DATA_BLOCK "DB22_DisplayData"   // DB22
{ S7_Optimized_Access := 'FALSE' }
AUTHOR : Robopac
VERSION : 0.0
// stored: AutoNumber false, IsOnlyStoredInLoadMemory false, IsWriteProtectedInAS false
   VAR RETAIN
      dbx0_0 : Bool := FALSE;   // Technoplat manual(Display): Table rotation forward
      dbx0_1 : Bool := FALSE;   // Technoplat manual(Display): Spool carriage upward
      dbx0_2 : Bool := FALSE;   // Technoplat manual(Display): Spool carriage downward
      dbx0_3 : Bool := FALSE;   // Technoplat manual(Display): Pressure plate upward/downward
      dbx0_4 : Bool := FALSE;   // Technoplat manual(Display): Pallet lifter upward/downward
      dbx0_5 : Bool := FALSE;   // Technoplat manual(Display): Rope unit open/close
      dbx0_6 : Bool := FALSE;   // Technoplat manual(Display): Prestretch
      dbx0_7 : Bool := FALSE;   // Technoplat manual(Display): Spool carriage to film broken position
      dbx1_0 : Bool := FALSE;   // Clamp manual(Display): Clamp upward/downward
      dbx1_1 : Bool := FALSE;   // Clamp manual(Display): Welder unit upward/downward
      dbx1_2 : Bool := FALSE;   // Clamp manual(Display): Welder contrast upward/downward
      dbx1_3 : Bool := FALSE;   // Clamp manual(Display): Clamp carriage forward/backward
      dbx1_4 : Bool := FALSE;   // Clamp manual(Display): Clamp open/close
      dbx1_5 : Bool := FALSE;   // Clamp manual(Display): Cut and welder arm forward/backward
      dbx1_6 : Bool := FALSE;   // Clamp manual(Display): Welder unit forward/backward
      dbx1_7 : Bool := FALSE;   // Clamp manual(Display):
      dbx2_0 : Bool := FALSE;   // Top manual(Display): Top carriage upward
      dbx2_1 : Bool := FALSE;   // Top manual(Display): Top carriage downward
      dbx2_2 : Bool := FALSE;   // Top manual(Display): Top carriage forward
      dbx2_3 : Bool := FALSE;   // Top manual(Display): Top carriage backward
      dbx2_4 : Bool := FALSE;   // Top manual(Display): Opening/closing clamp to pull top film
      dbx2_5 : Bool := FALSE;   // Top manual(Display): Opening/closing clamp to block top film
      dbx2_6 : Bool := FALSE;   // Top manual(Display): Top film cutter forward/backward
      dbx2_7 : Bool := FALSE;   // Top manual(Display): Arm rotation to phase 2 sensor for top
      dbx3_0 : Bool := FALSE;   // Technoplat manual (Display): Rotation to unload
      dbx3_1 : Bool := FALSE;   // Technoplat manual (Display): Rotation to 0
      dbx3_2 : Bool := FALSE;   // Technoplat manual (Display): Rotation to load
      dbx3_3 : Bool := FALSE;
      dbx3_4 : Bool := FALSE;   // Technoplat manual(Display): Rope unit lower open/close
      dbx3_5 : Bool := FALSE;
      dbx3_6 : Bool := FALSE;
      dbx3_7 : Bool := FALSE;
      dbx4_0 : Bool := FALSE;   // Conveyor manual(Display): CMD PRESSED
      dbx4_1 : Bool := FALSE;   // Conveyor manual(Display): Load CM [p18]
      dbx4_2 : Bool := FALSE;   // Conveyor manual(Display): Unload CM [p18]
      dbx4_3 : Bool := FALSE;   // Conveyor manual(Display): RESET ENCODER
      dbx4_4 : Bool := FALSE;   // Conveyor manual(Display): Load CM [Sysdata]
      dbx4_5 : Bool := FALSE;   // Conveyor manual(Display): [not used]
      dbx4_6 : Bool := FALSE;   // Conveyor manual(Display): CM backward slow
      dbx4_7 : Bool := FALSE;   // Conveyor manual(Display): CM forward slow
      dbb5 : Byte := 16#09;   // Conveyor manual operation
      dbx6_0 : Bool := FALSE;   // Manual Signal(Display): Pallet ready in infeed (Input)
      dbx6_1 : Bool := FALSE;   // Manual Signal(Display): Ready to receive pallet infeed (Output)
      dbx6_2 : Bool := FALSE;   // Manual Signal(Display): End of transfer pallet infeed (Output)
      dbx6_3 : Bool := FALSE;   // Manual Signal(Display): Pallet ready in outfeed (Output)
      dbx6_4 : Bool := FALSE;   // Manual Signal(Display): Ready to receive pallet outfeed (Input)
      dbx6_5 : Bool := FALSE;   // Manual Signal(Display): End of transfer pallet outfeed (Input)
      dbx6_6 : Bool := FALSE;   // Manual Signal(Display): Start wrapping signal (Input)
      dbx6_7 : Bool := FALSE;   // Manual Signal(Display): Customer conveyor stopped signal (Input)
      dbx7_0 : Bool := FALSE;   // Manual Signal(Display): Machine in position signal (Output)
      dbx7_1 : Bool := FALSE;   // Manual Signal(Display): Wrapp ended signal (Output)
      dbx7_2 : Bool := FALSE;   // Manual Signal(Display): Pallet in position for label
      dbx7_3 : Bool := TRUE;   // Manual Signal(Display): Label arm in position for pallet transfer
      dbx7_4 : Bool := FALSE;   // Manual Signal(Display): Label cycle ended
      dbx7_5 : Bool := FALSE;   // Manual Signal(Display): Label fault
      dbx7_6 : Bool := FALSE;
      dbx7_7 : Bool := FALSE;
      dbw8 : Int := 0;
      dbw10 : Int := 0;
      dbw12 : Int := 0;
      dbx14_0 : Bool := FALSE;   // Technoplat manual(Program): Table rotation forward
      dbx14_1 : Bool := FALSE;   // Technoplat manual(Program): Spool carriage upward
      dbx14_2 : Bool := FALSE;   // Technoplat manual(Program): Spool carriage downward
      dbx14_3 : Bool := FALSE;   // Technoplat manual(Program): Pressure plate downward
      dbx14_4 : Bool := FALSE;   // Technoplat manual(Program): Pressure plate upward
      dbx14_5 : Bool := FALSE;   // Technoplat manual(Program): Pallet lifter upward
      dbx14_6 : Bool := FALSE;   // Technoplat manual(Program): Pallet lifter downward
      dbx14_7 : Bool := FALSE;   // Technoplat manual(Program): Rope unit closing
      dbx15_0 : Bool := FALSE;   // Technoplat manual(Program): Rope unit opening
      dbx15_1 : Bool := FALSE;   // Technoplat manual(Program): Prestretch
      dbx15_2 : Bool := FALSE;   // Technoplat manual(Program): Spool carriage to film broken position
      dbx15_3 : Bool := FALSE;   // Technoplat manual(Program): Rope unit Lower closing
      dbx15_4 : Bool := FALSE;   // Technoplat manual(Program): Rope unit Lower opening
      dbx15_5 : Bool := FALSE;   // Technoplat manual(Program): CM Backward slow
      dbx15_6 : Bool := FALSE;   // Technoplat manual(Program): CM Forward slow
      dbx15_7 : Bool := FALSE;   // Technoplat manual(Program):
      dbx16_0 : Bool := FALSE;   // Clamp manual(Program): Clamp upward
      dbx16_1 : Bool := FALSE;   // Clamp manual(Program): Clamp downward
      dbx16_2 : Bool := FALSE;   // Clamp manual(Program): Welder unit upward
      dbx16_3 : Bool := FALSE;   // Clamp manual(Program): Welder unit downward
      dbx16_4 : Bool := FALSE;   // Clamp manual(Program): Welder contrast upward
      dbx16_5 : Bool := FALSE;   // Clamp manual(Program): Welder contrast downward
      dbx16_6 : Bool := FALSE;   // Clamp manual(Program): Clamp carriage forward
      dbx16_7 : Bool := FALSE;   // Clamp manual(Program): Clamp carriage backward
      dbx17_0 : Bool := FALSE;   // Clamp manual(Program): Clamp open
      dbx17_1 : Bool := FALSE;   // Clamp manual(Program): Clamp close
      dbx17_2 : Bool := FALSE;   // Clamp manual(Program): Cut and welder arm forward
      dbx17_3 : Bool := FALSE;   // Clamp manual(Program): Cut and welder arm backward
      dbx17_4 : Bool := FALSE;   // Clamp manual(Program): Welder unit forward
      dbx17_5 : Bool := FALSE;   // Clamp manual(Program): Welder unit backward
      dbx17_6 : Bool := FALSE;   // Clamp manual(Program):
      dbx17_7 : Bool := FALSE;   // Clamp manual(Program):
      dbx18_0 : Bool := FALSE;   // Top manual(Program): Top carriage upward
      dbx18_1 : Bool := FALSE;   // Top manual(Program): Top carriage downward
      dbx18_2 : Bool := FALSE;   // Top manual(Program): Top carriage forward
      dbx18_3 : Bool := FALSE;   // Top manual(Program): Top carriage backward
      dbx18_4 : Bool := FALSE;   // Top manual(Program): Opening clamp to pull top film
      dbx18_5 : Bool := FALSE;   // Top manual(Program): Closing clamp to pull top film
      dbx18_6 : Bool := FALSE;   // Top manual(Program): Opening clamp to block top film
      dbx18_7 : Bool := FALSE;   // Top manual(Program): Closing clamp to block top film
      dbx19_0 : Bool := FALSE;   // Top manual(Program): Top film cutter forward/backward
      dbx19_1 : Bool := FALSE;   // Top manual(Program): Arm rotation to phase 2 sensor for top
      dbx19_2 : Bool := FALSE;   // Technoplat manual(Program): Rotation to unload
      dbx19_3 : Bool := FALSE;   // Technoplat manual(Program): Rotation to 0
      dbx19_4 : Bool := FALSE;   // Technoplat manual(Program): Rotation to load
      dbx19_5 : Bool := FALSE;   // Top manual(Program):
      dbx19_6 : Bool := FALSE;   // Top manual(Program):
      dbx19_7 : Bool := FALSE;   // Top manual(Program):
      dbx20_0 : Bool := FALSE;   // Conveyor manual(Program): Load CM
      dbx20_1 : Bool := FALSE;   // Conveyor manual(Program): Unload CM
      dbx20_2 : Bool := FALSE;   // Conveyor manual(Program): CM backward
      dbx20_3 : Bool := FALSE;   // Conveyor manual(Program): Pos.1
      dbx20_4 : Bool := FALSE;   // Conveyor manual(Program): Pos.2
      dbx20_5 : Bool := FALSE;   // Conveyor manual(Program): Pos.3
      dbx20_6 : Bool := FALSE;   // Conveyor manual(Program): Pos.4
      dbx20_7 : Bool := FALSE;   // Conveyor manual(Program): Pos.5
      dbx21_0 : Bool := FALSE;   // Conveyor manual(Program): Pos.6
      dbx21_1 : Bool := FALSE;   // Conveyor manual(Program): Pos.7
      dbx21_2 : Bool := FALSE;   // Conveyor manual(Program): Pos.8
      dbx21_3 : Bool := FALSE;   // Conveyor manual(Program):
      dbx21_4 : Bool := FALSE;   // Conveyor manual(Program):
      dbx21_5 : Bool := FALSE;   // Conveyor manual(Program):
      dbx21_6 : Bool := FALSE;   // Conveyor manual(Program):
      dbx21_7 : Bool := FALSE;   // Conveyor manual(Program):
      dbx22_0 : Bool := FALSE;   // Manual Signal(Program): Pallet ready in infeed (Input)
      dbx22_1 : Bool := FALSE;   // Manual Signal(Program): Ready to receive pallet infeed (Output)
      dbx22_2 : Bool := FALSE;   // Manual Signal(Program): End of transfer pallet infeed (Output)
      dbx22_3 : Bool := FALSE;   // Manual Signal(Program): Pallet ready in outfeed (Output)
      dbx22_4 : Bool := FALSE;   // Manual Signal(Program): Ready to receive pallet outfeed (Input)
      dbx22_5 : Bool := FALSE;   // Manual Signal(Program): End of transfer pallet outfeed (Input)
      dbx22_6 : Bool := FALSE;   // Manual Signal(Program): Start wrapping (Input)
      dbx22_7 : Bool := FALSE;   // Manual Signal(Program): Customer conveyor stopped (Input)
      dbx23_0 : Bool := FALSE;   // Manual Signal(Program): Machine in position (Output)
      dbx23_1 : Bool := FALSE;   // Manual Signal(Program): Wrapp ended (Output)
      dbx23_2 : Bool := FALSE;   // Manual Signal(Program): Pallet ready for label
      dbx23_3 : Bool := TRUE;   // Manual Signal(Program): Label arm in position for pallet transfer
      dbx23_4 : Bool := FALSE;   // Manual Signal(Program): Label cycle ended
      dbx23_5 : Bool := FALSE;   // Manual Signal(Program): Label fault
      dbx23_6 : Bool := FALSE;
      dbx23_7 : Bool := FALSE;
      dbw24 : Int := 0;
      dbw26 : Int := 0;
      dbw28 : Int := 0;
      dbw30 : Int := 0;
      dbx32_0 : Bool := TRUE;   // Manual(Toggle bit): Pressure plate upward/downward (Technplat)
      dbx32_1 : Bool := TRUE;   // Manual(Toggle bit): Pallet lifter upward/downward (Technplat)
      dbx32_2 : Bool := FALSE;   // Manual(Toggle bit): Clamp upward/downward (Clamp)
      dbx32_3 : Bool := FALSE;   // Manual(Toggle bit): Welder unit upward/downward (Clamp)
      dbx32_4 : Bool := TRUE;   // Manual(Toggle bit): Welder contrast upward/downward (Clamp)
      dbx32_5 : Bool := FALSE;   // Manual(Toggle bit): Rope unit open/close (Technplat)
      dbx32_6 : Bool := FALSE;   // Manual(Toggle bit): Clamp open/close (Clamp)
      dbx32_7 : Bool := FALSE;   // Manual(Toggle bit): Cut and welder arm forward/backward (Clamp)
      dbx33_0 : Bool := TRUE;   // Manual(Toggle bit): Opening/closing clamp to pull top film (Top)
      dbx33_1 : Bool := TRUE;   // Manual(Toggle bit): Opening/closing clamp to block top film (Top)
      dbx33_2 : Bool := TRUE;   // Manual(Toggle bit): Welder unit forward/backward (Clamp)
      dbx33_3 : Bool := FALSE;   // Manual(Toggle bit): Clamp carriage forward/backward (Clamp)
      dbx33_4 : Bool := FALSE;   // Manual(Toggle bit): Rope unit lower open/close (Technplat)
      dbx33_5 : Bool := FALSE;   // Manual(Toggle bit):
      dbx33_6 : Bool := FALSE;   // Manual(Toggle bit):
      dbx33_7 : Bool := FALSE;   // Manual(Toggle bit):
      dbw34 : Int := 0;
      dbw36 : Int := 0;
      dbx38_0 : Bool := FALSE;   // Diagnostic signal conveyor: Pallet ready in infeed (input)
      dbx38_1 : Bool := TRUE;   // Diagnostic signal conveyor: Ready to receive pallet infeed (Output)
      dbx38_2 : Bool := FALSE;   // Diagnostic signal conveyor: End of transfer pallet infeed (Output)
      dbx38_3 : Bool := FALSE;   // Diagnostic signal conveyor: Ready to receive pallet in outfeed (Input)
      dbx38_4 : Bool := FALSE;   // Diagnostic signal conveyor: End of transfer pallet outfeed (Input)
      dbx38_5 : Bool := FALSE;   // Diagnostic signal conveyor: Pallet ready in outfeed (Output)
      dbx38_6 : Bool := FALSE;   // Diagnostic signal conveyor: Start wrapping (Input)
      dbx38_7 : Bool := FALSE;   // Diagnostic signal conveyor: Customer conveyor stopped (Input)
      dbx39_0 : Bool := FALSE;   // Diagnostic signal conveyor: Machine in position (Output)
      dbx39_1 : Bool := FALSE;   // Diagnostic signal conveyor: Wrapp ended (Output)
      dbx39_2 : Bool := FALSE;   // Diagnostic signal conveyor: Pallet ready for label
      dbx39_3 : Bool := TRUE;   // Diagnostic signal conveyor: Label arm in position for pallet transit
      dbx39_4 : Bool := FALSE;   // Diagnostic signal conveyor: Label cycle ended
      dbx39_5 : Bool := FALSE;   // Diagnostic signal conveyor: Label fault
      dbw40 : Int := 1;   // Machine status
      dbd42 : DInt := 4;   // Worked hours
      dbd46 : DInt := 95;   // Partial counter for wrapped pallet
      dbd50 : DInt := 163;   // Counter for wrapped pallet
      dbd54 : DInt := 0;
      dbw58 : Int := 21;   // Seconds for worked hours counter
      dbw60 : Int := 36;   // Minutes for worked hours counter
      dbw62 : Int := 0;   // Arm rotation speed (rpm)
      dbw64 : Int := 0;   // Arm rotation speed (rpm)
      dbw66 : Int := 15;   // Number of revolution done on last pallet
      dbw68 : Int := 777;   // Wrapping cycle time
      dbw70 : Int := 22482;   // Wrapping cycle + pallet transfer time
      dbw72 : Int := 10;   // Pallet per hour (Productivity)
      dbw74 : Int := 0;   // Film weight every wrapping cycle (g*10)
      dbw76 : Int := 0;   // Film force for film weight value
      dbw78 : Int := 0;   // Film prestretch for film weight value
      dbw80 : Int := 0;
      dbw82 : Int := 0;
      dbw84 : Int := 0;
      dbw86 : Int := 0;
      dbw88 : Int := 0;
      dbw90 : Int := 0;
      dbw92 : Int := 0;
      dbw94 : Int := 0;
      dbw96 : Int := 0;
      dbw98 : Int := 0;
   END_VAR
BEGIN
END_DATA_BLOCK

DATA_BLOCK "DB235_Program15"   // DB235
{ S7_Optimized_Access := 'FALSE' }
AUTHOR : Robopac
VERSION : 0.0
// stored: AutoNumber false, IsOnlyStoredInLoadMemory false, IsWriteProtectedInAS false
   VAR RETAIN
      Program15 { S7_SetPoint := 'True'} : "DatiProgramma";
   END_VAR
BEGIN
   Program15.Wrapping := TRUE;
   Program15.TopLenght := 500;
   Program15.TopRelease := 0;
   Program15.TopDown := 0;
   Program15.Top := 4;
   Program15.PressurePTime := 0;
   Program15.LifterTime := 0;
   Program15.RevOverContrast := 1;
   Program15.RopeEndCycle := 16#02;
   Program15.Spare4 := 16#01;
   Program15.RopeTime := 1500;
   Program15.RevOverClamp := 1;
   Program15.FilmForceFinalRev := 10;
   Program15.FilmPrestretchFinalRev := 100;
   Program15.ArmSpeed := 100;
   Program15.CarriageDown4Top := 500;
   Program15.TopDownTime := 1500;
   Program15.LapsUnderTop := 0;
   Program15.Spare6 := 0;
   Program15.Spare7 := 0;
   Program15.Spare8 := 0;
   Program15.Spare9 := 0;
   Program15.Spare10 := 0;
   Program15.Spare11 := 0;
   Program15.Spare12 := 0;
   Program15.Overlap0_1 := 0;
   Program15.Height1 := 130;
   Program15.Landmark1 := FALSE;
   Program15.Lifter1 := FALSE;
   Program15.SpareBit1H1 := FALSE;
   Program15.Airblower1 := TRUE;
   Program15.NextStep1 := TRUE;
   Program15.PressureP1 := TRUE;
   Program15.SpareByte2H1 := 16#00;
   Program15.Revolution1 := 1;
   Program15.RopeUnit1_1 := 16#01;
   Program15.RopeUnit1_2 := 16#01;
   Program15.FilmForce1 := 5;
   Program15.FilmPrestretch1 := 200;
   Program15.Spare3H1 := 0;
   Program15.Spare49 := 0;
   Program15.Spare50 := 0;
   Program15.Spare51 := 0;
   Program15.Spare52 := 0;
   Program15.Spare53 := 0;
   Program15.Overlap1_2 := 0;
   Program15.Height2 := 50;
   Program15.Landmark2 := FALSE;
   Program15.Lifter2 := FALSE;
   Program15.SpareBit1H2 := FALSE;
   Program15.Airblower2 := TRUE;
   Program15.NextStep2 := TRUE;
   Program15.PressureP2 := TRUE;
   Program15.SpareByte2H2 := 16#00;
   Program15.Revolution2 := 1;
   Program15.RopeUnit2_1 := 16#01;
   Program15.RopeUnit2_2 := 16#01;
   Program15.FilmForce2 := 20;
   Program15.FilmPrestretch2 := 200;
   Program15.Spare3H2 := 0;
   Program15.Spare54 := 0;
   Program15.Spare55 := 0;
   Program15.Spare56 := 0;
   Program15.Spare57 := 0;
   Program15.Spare58 := 0;
   Program15.Overlap2_3 := 100;
   Program15.Height3 := -50;
   Program15.Landmark3 := TRUE;
   Program15.Lifter3 := FALSE;
   Program15.SpareBit1H3 := FALSE;
   Program15.Airblower3 := TRUE;
   Program15.NextStep3 := TRUE;
   Program15.PressureP3 := TRUE;
   Program15.SpareByte2H3 := 16#00;
   Program15.Revolution3 := 2;
   Program15.RopeUnit3_1 := 16#01;
   Program15.RopeUnit3_2 := 16#01;
   Program15.FilmForce3 := 30;
   Program15.FilmPrestretch3 := 200;
   Program15.Spare3H3 := 0;
   Program15.Spare59 := 0;
   Program15.Spare60 := 0;
   Program15.Spare61 := 380;
   Program15.Spare62 := 2800;
   Program15.Spare63 := 0;
   Program15.Overlap3_4 := 100;
   Program15.Height4 := 100;
   Program15.Landmark4 := FALSE;
   Program15.Lifter4 := FALSE;
   Program15.SpareBit1H4 := FALSE;
   Program15.Airblower4 := TRUE;
   Program15.NextStep4 := TRUE;
   Program15.PressureP4 := TRUE;
   Program15.SpareByte2H4 := 16#00;
   Program15.Revolution4 := 3;
   Program15.RopeUnit4_1 := 16#02;
   Program15.RopeUnit4_2 := 16#02;
   Program15.FilmForce4 := 30;
   Program15.FilmPrestretch4 := 200;
   Program15.Spare3H4 := 0;
   Program15.Spare64 := 0;
   Program15.Spare65 := 0;
   Program15.Spare66 := 0;
   Program15.Spare67 := 0;
   Program15.Spare68 := 0;
   Program15.Overlap4_5 := 0;
   Program15.Height5 := 50;
   Program15.Landmark5 := FALSE;
   Program15.Lifter5 := FALSE;
   Program15.SpareBit1H5 := FALSE;
   Program15.Airblower5 := TRUE;
   Program15.NextStep5 := FALSE;
   Program15.PressureP5 := FALSE;
   Program15.SpareByte2H5 := 16#00;
   Program15.Revolution5 := 1;
   Program15.RopeUnit5_1 := 16#01;
   Program15.RopeUnit5_2 := 16#01;
   Program15.FilmForce5 := 30;
   Program15.FilmPrestretch5 := 200;
   Program15.Spare3H5 := 0;
   Program15.Spare69 := 0;
   Program15.Spare70 := 0;
   Program15.Spare71 := 0;
   Program15.Spare72 := 0;
   Program15.Spare73 := 0;
   Program15.Overlap5_6 := 100;
   Program15.Height6 := 50;
   Program15.Landmark6 := FALSE;
   Program15.Lifter6 := FALSE;
   Program15.SpareBit1H6 := FALSE;
   Program15.Airblower6 := TRUE;
   Program15.NextStep6 := FALSE;
   Program15.PressureP6 := FALSE;
   Program15.SpareByte2H6 := 16#00;
   Program15.Revolution6 := 2;
   Program15.RopeUnit6_1 := 16#02;
   Program15.RopeUnit6_2 := 16#01;
   Program15.FilmForce6 := 20;
   Program15.FilmPrestretch6 := 200;
   Program15.Spare3H6 := 0;
   Program15.Spare74 := 0;
   Program15.Spare75 := 0;
   Program15.Spare76 := 0;
   Program15.Spare77 := 0;
   Program15.Spare78 := 0;
   Program15.Overlap6_7 := 0;
   Program15.Height7 := 0;
   Program15.Landmark7 := FALSE;
   Program15.Lifter7 := FALSE;
   Program15.SpareBit1H7 := FALSE;
   Program15.Airblower7 := FALSE;
   Program15.NextStep7 := TRUE;
   Program15.PressureP7 := FALSE;
   Program15.SpareByte2H7 := 16#00;
   Program15.Revolution7 := 1;
   Program15.RopeUnit7_1 := 16#01;
   Program15.RopeUnit7_2 := 16#01;
   Program15.FilmForce7 := 0;
   Program15.FilmPrestretch7 := 100;
   Program15.Spare3H7 := 0;
   Program15.Spare79 := 0;
   Program15.Spare80 := 0;
   Program15.Spare81 := 0;
   Program15.Spare82 := 0;
   Program15.Spare83 := 0;
   Program15.Overlap7_8 := 0;
   Program15.Height8 := 0;
   Program15.Landmark8 := FALSE;
   Program15.Lifter8 := FALSE;
   Program15.SpareBit1H8 := FALSE;
   Program15.Airblower8 := FALSE;
   Program15.NextStep8 := TRUE;
   Program15.PressureP8 := FALSE;
   Program15.SpareByte2H8 := 16#00;
   Program15.Revolution8 := 1;
   Program15.RopeUnit8_1 := 16#01;
   Program15.RopeUnit8_2 := 16#01;
   Program15.FilmForce8 := 0;
   Program15.FilmPrestretch8 := 100;
   Program15.Spare3H8 := 0;
   Program15.Spare84 := 0;
   Program15.Spare85 := 0;
   Program15.Spare86 := 0;
   Program15.Spare87 := 0;
   Program15.Spare88 := 0;
   Program15.Overlap8_9 := 0;
   Program15.Height9 := 0;
   Program15.Landmark9 := FALSE;
   Program15.Lifter9 := FALSE;
   Program15.SpareBit1H9 := FALSE;
   Program15.Airblower9 := FALSE;
   Program15.NextStep9 := TRUE;
   Program15.PressureP9 := FALSE;
   Program15.SpareByte2H9 := 16#00;
   Program15.Revolution9 := 1;
   Program15.RopeUnit9_1 := 16#01;
   Program15.RopeUnit9_2 := 16#01;
   Program15.FilmForce9 := 0;
   Program15.FilmPrestretch9 := 100;
   Program15.Spare3H9 := 0;
   Program15.Spare89 := 0;
   Program15.Spare90 := 0;
   Program15.Spare91 := 0;
   Program15.Spare92 := 0;
   Program15.Spare93 := 0;
   Program15.Overlap9_10 := 0;
   Program15.Height10 := 0;
   Program15.Landmark10 := FALSE;
   Program15.Lifter10 := FALSE;
   Program15.SpareBit1H10 := FALSE;
   Program15.Airblower10 := FALSE;
   Program15.NextStep10 := FALSE;
   Program15.PressureP10 := FALSE;
   Program15.SpareByte2H10 := 16#00;
   Program15.Revolution10 := 1;
   Program15.RopeUnit10_1 := 16#01;
   Program15.RopeUnit10_2 := 16#01;
   Program15.FilmForce10 := 0;
   Program15.FilmPrestretch10 := 100;
   Program15.Spare3H10 := 0;
   Program15.Spare94 := 0;
   Program15.Spare95 := 0;
   Program15.Spare96 := 0;
   Program15.Spare97 := 0;
   Program15.Spare98 := 0;
   Program15.Overlap10_11 := 0;
   Program15.Height11 := 0;
   Program15.Landmark11 := FALSE;
   Program15.Lifter11 := FALSE;
   Program15.SpareBit1H11 := FALSE;
   Program15.Airblower11 := FALSE;
   Program15.NextStep11 := TRUE;
   Program15.PressureP11 := FALSE;
   Program15.SpareByte2H11 := 16#00;
   Program15.Revolution11 := 1;
   Program15.RopeUnit11_1 := 16#01;
   Program15.RopeUnit11_2 := 16#01;
   Program15.FilmForce11 := 0;
   Program15.FilmPrestretch11 := 100;
   Program15.Spare3H11 := 0;
   Program15.Spare99 := 0;
   Program15.Spare100 := 0;
   Program15.Spare101 := 0;
   Program15.Spare102 := 0;
   Program15.Spare103 := 0;
   Program15.Overlap11_12 := 0;
   Program15.Height12 := 0;
   Program15.Landmark12 := FALSE;
   Program15.Lifter12 := FALSE;
   Program15.SpareBit1H12 := FALSE;
   Program15.Airblower12 := FALSE;
   Program15.NextStep12 := FALSE;
   Program15.PressureP12 := FALSE;
   Program15.SpareByte2H12 := 16#00;
   Program15.Revolution12 := 1;
   Program15.RopeUnit12_1 := 16#01;
   Program15.RopeUnit12_2 := 16#01;
   Program15.FilmForce12 := 0;
   Program15.FilmPrestretch12 := 100;
   Program15.Spare3H12 := 0;
   Program15.Spare104 := 0;
   Program15.Spare105 := 0;
   Program15.Spare106 := 0;
   Program15.Spare107 := 0;
   Program15.Spare108 := 0;
END_DATA_BLOCK

DATA_BLOCK "DB23_AlarmProgram"   // DB23
{ S7_Optimized_Access := 'FALSE' }
AUTHOR : Robopac
VERSION : 0.0
// stored: AutoNumber false, IsOnlyStoredInLoadMemory false, IsWriteProtectedInAS false
   VAR RETAIN
      dbx0_0 : Bool := FALSE;   // Alarm 1: Pressure switch (Technoplat)
      dbx0_1 : Bool := FALSE;   // Alarm 2: Door open request (Technoplat)
      dbx0_2 : Bool := FALSE;   // Alarm 3: Emergency push button (Technoplat)
      dbx0_3 : Bool := FALSE;   // Alarm 4: Thermic alarm (Technoplat)
      dbx0_4 : Bool := FALSE;   // Alarm 5: Fault inverters (Technoplat)
      dbx0_5 : Bool := FALSE;   // Alarm 6: Motor start missing (Technoplat)
      dbx0_6 : Bool := FALSE;   // Alarm 7: Stop cycle by operator (Technoplat)
      dbx0_7 : Bool := FALSE;   // Alarm 8: Film ended or broken (Technoplat)
      dbx1_0 : Bool := FALSE;   // Alarm 9: Machine table not in phase (Technoplat)
      dbx1_1 : Bool := FALSE;   // Alarm 10: The spool carriage encoder is not running (Technoplat)
      dbx1_2 : Bool := FALSE;   // Alarm 11: Table encoder not working well
      dbx1_3 : Bool := FALSE;   // Alarm 12: Overspeed for table rotation (Technoplat)
      dbx1_4 : Bool := FALSE;   // Alarm 13: Phase table sensor lost (Technoplat)
      dbx1_5 : Bool := FALSE;   // Alarm 14: table deceleration not correct (Technoplat)
      dbx1_6 : Bool := FALSE;   // Alarm 15: Pressure plate not up (Pressure plate)
      dbx1_7 : Bool := FALSE;   // Alarm 16: Timeout for pressure plate upward/downward (Pressure plate)
      dbx2_0 : Bool := FALSE;   // Alarm 17: Pallet lifter not down (Lifter)
      dbx2_1 : Bool := FALSE;   // Alarm 18: Timeout for pallet lifter upward/downward (Lifter)
      dbx2_2 : Bool := FALSE;   // Alarm 19: Wrong data program for the pallet on the machine (Technoplat)
      dbx2_3 : Bool := FALSE;   // Alarm 20: Sysdata error (Technoplat)
      dbx2_4 : Bool := FALSE;   // Alarm 21: Spool carriage not down (Technoplat)
      dbx2_5 : Bool := FALSE;   // Alarm 22: Pressure plate positioning lost during rotation
      dbx2_6 : Bool := FALSE;   // Alarm 23:
      dbx2_7 : Bool := FALSE;   // Alarm 24: Emergency on infeed safety barrier (Barrier)
      dbx3_0 : Bool := FALSE;   // Alarm 25: Emergency on outfeed safety barrier (Barrier)
      dbx3_1 : Bool := FALSE;   // Alarm 26: Safety barrier excluded in automatic mode (Barrier)
      dbx3_2 : Bool := FALSE;   // Alarm 27: Timeout for rope unit open/close (Rope unit)
      dbx3_3 : Bool := FALSE;   // Alarm 28: Timeout for full rope unit open/close (Rope unit)
      dbx3_4 : Bool := FALSE;   // Alarm 29:
      dbx3_5 : Bool := FALSE;   // Alarm 30: Profinet communication error
      dbx3_6 : Bool := FALSE;   // Alarm 31: Modbus communication error
      dbx3_7 : Bool := FALSE;   // Alarm 32:
      dbx4_0 : Bool := FALSE;   // Alarm 33: Pallet positioning released during table rotation (Conveyor
      dbx4_1 : Bool := FALSE;   // Alarm 34: Pallet in transit in infeed (Conveyor)
      dbx4_2 : Bool := FALSE;   // Alarm 35: Pallet in transit in outfeed (Conveyor)
      dbx4_3 : Bool := FALSE;   // Alarm 36: Wrong pallet positioning (Conveyor)
      dbx4_4 : Bool := FALSE;   // Alarm 37: Infeed ring rotation control engaged (Conveyor)
      dbx4_5 : Bool := FALSE;   // Alarm 38: Outfeed ring rotation control engaged (Conveyor)
      dbx4_6 : Bool := FALSE;   // Alarm 39: Technoplat table not in load phase
      dbx4_7 : Bool := FALSE;   // Alarm 40: Technoplat table not in unload phase
      dbx5_0 : Bool := FALSE;   // Alarm 41: Contrast carriage not back
      dbx5_1 : Bool := FALSE;   // Alarm 42: Timeout contrast carriage forward/backward
      dbx5_2 : Bool := FALSE;   // Alarm 43: Clamp not closed (Clamp)
      dbx5_3 : Bool := FALSE;   // Alarm 44: Welder contrast not down (Clamp)
      dbx5_4 : Bool := FALSE;   // Alarm 45: Welder unit not down (Clamp)
      dbx5_5 : Bool := FALSE;   // Alarm 46: Clamp not down (Clamp)
      dbx5_6 : Bool := FALSE;   // Alarm 47: Welder contrast not up (Clamp)
      dbx5_7 : Bool := FALSE;   // Alarm 48: Timeout for clamp open/close (Clamp)
      dbx6_0 : Bool := FALSE;   // Alarm 49: Timeout for clamp upward/downward (Clamp)
      dbx6_1 : Bool := FALSE;   // Alarm 50: Timeout for welder contrast upward/downward (Clamp)
      dbx6_2 : Bool := FALSE;   // Alarm 51: Timeout for welder unit upward/downward (Clamp)
      dbx6_3 : Bool := FALSE;   // Alarm 52: Check the welder circuit (Clamp)
      dbx6_4 : Bool := FALSE;   // Alarm 53: Welder and cut unit not backward (Clamp)
      dbx6_5 : Bool := FALSE;   // Alarm 54: Timeout for welder and cut unit forward/backward (Clamp)
      dbx6_6 : Bool := FALSE;   // Alarm 55: Timeout for clamp carriage forward/backward (Clamp)
      dbx6_7 : Bool := FALSE;   // Alarm 56: Clamp carriage not backward (Clamp)
      dbx7_0 : Bool := FALSE;   // Alarm 57: Top carriage not up (Top)
      dbx7_1 : Bool := FALSE;   // Alarm 58: Top carriage not backward (Top)
      dbx7_2 : Bool := FALSE;   // Alarm 59: Top cutter not backward (Top)
      dbx7_3 : Bool := FALSE;   // Alarm 60: Clamp to pull top film not open (Top)
      dbx7_4 : Bool := FALSE;   // Alarm 61: Clamp to block top film not closed (Top)
      dbx7_5 : Bool := FALSE;   // Alarm 62: Top carriage not in position (Top)
      dbx7_6 : Bool := FALSE;   // Alarm 63: Top carriage not inside top film cut area (Top)
      dbx7_7 : Bool := FALSE;   // Alarm 64: Safety for top carriage position (Top)
      dbx8_0 : Bool := FALSE;   // Alarm 65: Timeout for top cutter (Top)
      dbx8_1 : Bool := FALSE;   // Alarm 66: Timeout for clamp to pull top film (Top)
      dbx8_2 : Bool := FALSE;   // Alarm 67: Timeout for clamp to block top film (Top)
      dbx8_3 : Bool := FALSE;   // Alarm 68: Top film ended or broken (Top)
      dbx8_4 : Bool := FALSE;   // Alarm 69: Infeed safety for top carriage up/down (Top)
      dbx8_5 : Bool := FALSE;   // Alarm 70: Outfeed safety for top carriage up/down (Top)
      dbx8_6 : Bool := FALSE;   // Alarm 71: Clamp to blok top film not open (Top)
      dbx8_7 : Bool := FALSE;   // Alarm 72: Top rele' brake broken (Top)
      dbx9_0 : Bool := FALSE;   // Alarm 73: Top not in position (Top inside signal)
      dbx9_1 : Bool := FALSE;   // Alarm 74: LIFTER POS.2 EXTRASTROKE UP
      dbx9_2 : Bool := FALSE;   // Alarm 75: LIFTER POS.2 FOOT SAFETY
      dbx9_3 : Bool := FALSE;   // Alarm 76: LIFTER POS.2 TIMEOUT CONVEYOR
      dbx9_4 : Bool := FALSE;   // Alarm 77: LIFTER POS.2 TIMEOUT UPSTROKE
      dbx9_5 : Bool := FALSE;   // Alarm 78: LIFTER POS.2 TIMEOUT DOWNSTROKE
      dbx9_6 : Bool := FALSE;   // Alarm 79: LABEL FAULT
      dbx9_7 : Bool := FALSE;   // Alarm 80: Label not in home position with table rotation
      dbx10_0 : Bool := FALSE;   // Alarm 81: Fire door not open during pallet transit
      dbx10_1 : Bool := FALSE;   // Alarm 82:
      dbx10_2 : Bool := FALSE;   // Alarm 83:
      dbx10_3 : Bool := FALSE;   // Alarm 84:
      dbx10_4 : Bool := FALSE;   // Alarm 85:
      dbx10_5 : Bool := FALSE;   // Alarm 86:
      dbx10_6 : Bool := FALSE;   // Alarm 87:
      dbx10_7 : Bool := FALSE;   // Alarm 88:
      dbx11_0 : Bool := FALSE;   // Alarm 89:
      dbx11_1 : Bool := FALSE;   // Alarm 90:
      dbx11_2 : Bool := FALSE;   // Alarm 91:
      dbx11_3 : Bool := FALSE;   // Alarm 92:
      dbx11_4 : Bool := FALSE;   // Alarm 93:
      dbx11_5 : Bool := FALSE;   // Alarm 94:
      dbx11_6 : Bool := FALSE;   // Alarm 95:
      dbx11_7 : Bool := FALSE;   // Alarm 96:
      dbx12_0 : Bool := FALSE;   // Alarm 97:
      dbx12_1 : Bool := FALSE;   // Alarm 98:
      dbx12_2 : Bool := FALSE;   // Alarm 99:
      dbx12_3 : Bool := FALSE;   // Alarm 100:
      dbx12_4 : Bool := FALSE;   // Alarm 101:
      dbx12_5 : Bool := FALSE;   // Alarm 102:
      dbx12_6 : Bool := FALSE;   // Alarm 103:
      dbx12_7 : Bool := FALSE;   // Alarm 104:
      dbx13_0 : Bool := FALSE;   // Alarm 105:
      dbx13_1 : Bool := FALSE;   // Alarm 106:
      dbx13_2 : Bool := FALSE;   // Alarm 107:
      dbx13_3 : Bool := FALSE;   // Alarm 108:
      dbx13_4 : Bool := FALSE;   // Alarm 109:
      dbx13_5 : Bool := FALSE;   // Alarm 110:
      dbx13_6 : Bool := FALSE;   // Alarm 111:
      dbx13_7 : Bool := FALSE;   // Alarm 112:
      dbx14_0 : Bool := FALSE;   // Alarm 113:
      dbx14_1 : Bool := FALSE;   // Alarm 114:
      dbx14_2 : Bool := FALSE;   // Alarm 115:
      dbx14_3 : Bool := FALSE;   // Alarm 116:
      dbx14_4 : Bool := FALSE;   // Alarm 117:
      dbx14_5 : Bool := FALSE;   // Alarm 118:
      dbx14_6 : Bool := FALSE;   // Alarm 119:
      dbx14_7 : Bool := FALSE;   // Alarm 120:
      dbx15_0 : Bool := FALSE;   // Alarm 121:
      dbx15_1 : Bool := FALSE;   // Alarm 122:
      dbx15_2 : Bool := FALSE;   // Alarm 123:
      dbx15_3 : Bool := FALSE;   // Alarm 124:
      dbx15_4 : Bool := FALSE;   // Alarm 125:
      dbx15_5 : Bool := FALSE;   // Alarm 126:
      dbx15_6 : Bool := FALSE;   // Alarm 127:
      dbx15_7 : Bool := FALSE;   // Alarm 128:
      dbx16_0 : Bool := FALSE;   // Alarm 129:
      dbx16_1 : Bool := FALSE;   // Alarm 130:
      dbx16_2 : Bool := FALSE;   // Alarm 131:
      dbx16_3 : Bool := FALSE;   // Alarm 132:
      dbx16_4 : Bool := FALSE;   // Alarm 133:
      dbx16_5 : Bool := FALSE;   // Alarm 134:
      dbx16_6 : Bool := FALSE;   // Alarm 135:
      dbx16_7 : Bool := FALSE;   // Alarm 136:
      dbx17_0 : Bool := FALSE;   // Alarm 137:
      dbx17_1 : Bool := FALSE;   // Alarm 138:
      dbx17_2 : Bool := FALSE;   // Alarm 139:
      dbx17_3 : Bool := FALSE;   // Alarm 140:
      dbx17_4 : Bool := FALSE;   // Alarm 141:
      dbx17_5 : Bool := FALSE;   // Alarm 142:
      dbx17_6 : Bool := FALSE;   // Alarm 143:
      dbx17_7 : Bool := FALSE;   // Alarm 144:
      dbx18_0 : Bool := FALSE;   // Alarm 145:
      dbx18_1 : Bool := FALSE;   // Alarm 146:
      dbx18_2 : Bool := FALSE;   // Alarm 147:
      dbx18_3 : Bool := FALSE;   // Alarm 148:
      dbx18_4 : Bool := FALSE;   // Alarm 149:
      dbx18_5 : Bool := FALSE;   // Alarm 150:
      dbx18_6 : Bool := FALSE;   // Alarm 151:
      dbx18_7 : Bool := FALSE;   // Alarm 152:
      dbx19_0 : Bool := FALSE;   // Alarm 153:
      dbx19_1 : Bool := FALSE;   // Alarm 154:
      dbx19_2 : Bool := FALSE;   // Alarm 155:
      dbx19_3 : Bool := FALSE;   // Alarm 156:
      dbx19_4 : Bool := FALSE;   // Alarm 157:
      dbx19_5 : Bool := FALSE;   // Alarm 158:
      dbx19_6 : Bool := FALSE;   // Alarm 159:
      dbx19_7 : Bool := FALSE;   // Alarm 160:
      dbx20_0 : Bool := FALSE;   // Alarm 161:
      dbx20_1 : Bool := FALSE;   // Alarm 162:
      dbx20_2 : Bool := FALSE;   // Alarm 163:
      dbx20_3 : Bool := FALSE;   // Alarm 164:
      dbx20_4 : Bool := FALSE;   // Alarm 165:
      dbx20_5 : Bool := FALSE;   // Alarm 166:
      dbx20_6 : Bool := FALSE;   // Alarm 167:
      dbx20_7 : Bool := FALSE;   // Alarm 168:
      dbx21_0 : Bool := FALSE;   // Alarm 169:
      dbx21_1 : Bool := FALSE;   // Alarm 170:
      dbx21_2 : Bool := FALSE;   // Alarm 171:
      dbx21_3 : Bool := FALSE;   // Alarm 172:
      dbx21_4 : Bool := FALSE;   // Alarm 173:
      dbx21_5 : Bool := FALSE;   // Alarm 174:
      dbx21_6 : Bool := FALSE;   // Alarm 175:
      dbx21_7 : Bool := FALSE;   // Alarm 176:
      dbx22_0 : Bool := FALSE;   // Alarm 177:
      dbx22_1 : Bool := FALSE;   // Alarm 178:
      dbx22_2 : Bool := FALSE;   // Alarm 179:
      dbx22_3 : Bool := FALSE;   // Alarm 180:
      dbx22_4 : Bool := FALSE;   // Alarm 181:
      dbx22_5 : Bool := FALSE;   // Alarm 182:
      dbx22_6 : Bool := FALSE;   // Alarm 183:
      dbx22_7 : Bool := FALSE;   // Alarm 184:
      dbx23_0 : Bool := FALSE;   // Alarm 185:
      dbx23_1 : Bool := FALSE;   // Alarm 186:
      dbx23_2 : Bool := FALSE;   // Alarm 187:
      dbx23_3 : Bool := FALSE;   // Alarm 188:
      dbx23_4 : Bool := FALSE;   // Alarm 189:
      dbx23_5 : Bool := FALSE;   // Alarm 190:
      dbx23_6 : Bool := FALSE;   // Alarm 191:
      dbx23_7 : Bool := FALSE;   // Alarm 192:
      dbx24_0 : Bool := FALSE;   // Alarm 193:
      dbx24_1 : Bool := FALSE;   // Alarm 194:
      dbx24_2 : Bool := FALSE;   // Alarm 195:
      dbx24_3 : Bool := FALSE;   // Alarm 196:
      dbx24_4 : Bool := FALSE;   // Alarm 197:
      dbx24_5 : Bool := FALSE;   // Alarm 198:
      dbx24_6 : Bool := FALSE;   // Alarm 199:
      dbx24_7 : Bool := FALSE;   // Alarm 200:
      dbx25_0 : Bool := FALSE;   // Alarm 201:
      dbx25_1 : Bool := FALSE;   // Alarm 202:
      dbx25_2 : Bool := FALSE;   // Alarm 203:
      dbx25_3 : Bool := FALSE;   // Alarm 204:
      dbx25_4 : Bool := FALSE;   // Alarm 205:
      dbx25_5 : Bool := FALSE;   // Alarm 206:
      dbx25_6 : Bool := FALSE;   // Alarm 207:
      dbx25_7 : Bool := FALSE;   // Alarm 208:
      dbx26_0 : Bool := FALSE;   // Warning 1: %10 Prestretch film on spool carriage (Technoplat)
      dbx26_1 : Bool := FALSE;   // Warning 2:
      dbx26_2 : Bool := FALSE;   // Warning 3: Request to reset encoder on spool carriage (Technoplat)
      dbx26_3 : Bool := FALSE;   // Warning 4:
      dbx26_4 : Bool := FALSE;   // Warning 5: Request to reset encoder on table rotation (Technoplat)
      dbx26_5 : Bool := FALSE;   // Warning 6:
      dbx26_6 : Bool := FALSE;   // Warning 7:
      dbx26_7 : Bool := FALSE;   // Warning 8: Fire door closing request
      dbx27_0 : Bool := FALSE;   // Warning 9: Timeout for door opening
      dbx27_1 : Bool := FALSE;   // Warning 10:
      dbx27_2 : Bool := FALSE;   // Warning 11:
      dbx27_3 : Bool := FALSE;   // Warning 12:
      dbx27_4 : Bool := FALSE;   // Warning 13:
      dbx27_5 : Bool := FALSE;   // Warning 14:
      dbx27_6 : Bool := FALSE;   // Warning 15:
      dbx27_7 : Bool := FALSE;   // Warning 16:
      dbx28_0 : Bool := FALSE;   // Warning 17:
      dbx28_1 : Bool := FALSE;   // Warning 18:
      dbx28_2 : Bool := FALSE;   // Warning 19:
      dbx28_3 : Bool := FALSE;   // Warning 20:
      dbx28_4 : Bool := FALSE;   // Warning 21:
      dbx28_5 : Bool := FALSE;   // Warning 22:
      dbx28_6 : Bool := FALSE;   // Warning 23:
      dbx28_7 : Bool := FALSE;   // Warning 24:
      dbx29_0 : Bool := FALSE;   // Warning 25:
      dbx29_1 : Bool := FALSE;   // Warning 26:
      dbx29_2 : Bool := FALSE;   // Warning 27:
      dbx29_3 : Bool := FALSE;   // Warning 28:
      dbx29_4 : Bool := FALSE;   // Warning 29:
      dbx29_5 : Bool := FALSE;   // Warning 30:
      dbx29_6 : Bool := FALSE;   // Warning 31:
      dbx29_7 : Bool := FALSE;   // Warning 32:
   END_VAR
BEGIN
END_DATA_BLOCK

DATA_BLOCK "DB240_Program10"   // DB240
{ S7_Optimized_Access := 'FALSE' }
AUTHOR : Robopac
VERSION : 0.0
// stored: AutoNumber false, IsOnlyStoredInLoadMemory false, IsWriteProtectedInAS false
   VAR RETAIN
      Program10 { S7_SetPoint := 'True'} : "DatiProgramma";
   END_VAR
BEGIN
   Program10.Wrapping := TRUE;
   Program10.TopLenght := 500;
   Program10.TopRelease := 0;
   Program10.TopDown := 0;
   Program10.Top := 4;
   Program10.PressurePTime := 0;
   Program10.LifterTime := 0;
   Program10.RevOverContrast := 1;
   Program10.RopeEndCycle := 16#02;
   Program10.Spare4 := 16#01;
   Program10.RopeTime := 1500;
   Program10.RevOverClamp := 1;
   Program10.FilmForceFinalRev := 10;
   Program10.FilmPrestretchFinalRev := 100;
   Program10.ArmSpeed := 100;
   Program10.CarriageDown4Top := 500;
   Program10.TopDownTime := 1500;
   Program10.LapsUnderTop := 0;
   Program10.Spare6 := 0;
   Program10.Spare7 := 0;
   Program10.Spare8 := 0;
   Program10.Spare9 := 0;
   Program10.Spare10 := 0;
   Program10.Spare11 := 0;
   Program10.Spare12 := 0;
   Program10.Overlap0_1 := 0;
   Program10.Height1 := 130;
   Program10.Landmark1 := FALSE;
   Program10.Lifter1 := FALSE;
   Program10.SpareBit1H1 := FALSE;
   Program10.Airblower1 := TRUE;
   Program10.NextStep1 := TRUE;
   Program10.PressureP1 := TRUE;
   Program10.SpareByte2H1 := 16#00;
   Program10.Revolution1 := 1;
   Program10.RopeUnit1_1 := 16#01;
   Program10.RopeUnit1_2 := 16#01;
   Program10.FilmForce1 := 5;
   Program10.FilmPrestretch1 := 200;
   Program10.Spare3H1 := 0;
   Program10.Spare49 := 0;
   Program10.Spare50 := 0;
   Program10.Spare51 := 0;
   Program10.Spare52 := 0;
   Program10.Spare53 := 0;
   Program10.Overlap1_2 := 0;
   Program10.Height2 := 50;
   Program10.Landmark2 := FALSE;
   Program10.Lifter2 := FALSE;
   Program10.SpareBit1H2 := FALSE;
   Program10.Airblower2 := TRUE;
   Program10.NextStep2 := TRUE;
   Program10.PressureP2 := TRUE;
   Program10.SpareByte2H2 := 16#00;
   Program10.Revolution2 := 1;
   Program10.RopeUnit2_1 := 16#01;
   Program10.RopeUnit2_2 := 16#01;
   Program10.FilmForce2 := 20;
   Program10.FilmPrestretch2 := 200;
   Program10.Spare3H2 := 0;
   Program10.Spare54 := 0;
   Program10.Spare55 := 0;
   Program10.Spare56 := 0;
   Program10.Spare57 := 0;
   Program10.Spare58 := 0;
   Program10.Overlap2_3 := 100;
   Program10.Height3 := -50;
   Program10.Landmark3 := TRUE;
   Program10.Lifter3 := FALSE;
   Program10.SpareBit1H3 := FALSE;
   Program10.Airblower3 := TRUE;
   Program10.NextStep3 := TRUE;
   Program10.PressureP3 := TRUE;
   Program10.SpareByte2H3 := 16#00;
   Program10.Revolution3 := 2;
   Program10.RopeUnit3_1 := 16#01;
   Program10.RopeUnit3_2 := 16#01;
   Program10.FilmForce3 := 30;
   Program10.FilmPrestretch3 := 200;
   Program10.Spare3H3 := 0;
   Program10.Spare59 := 0;
   Program10.Spare60 := 0;
   Program10.Spare61 := 380;
   Program10.Spare62 := 2800;
   Program10.Spare63 := 0;
   Program10.Overlap3_4 := 100;
   Program10.Height4 := 100;
   Program10.Landmark4 := FALSE;
   Program10.Lifter4 := FALSE;
   Program10.SpareBit1H4 := FALSE;
   Program10.Airblower4 := TRUE;
   Program10.NextStep4 := TRUE;
   Program10.PressureP4 := TRUE;
   Program10.SpareByte2H4 := 16#00;
   Program10.Revolution4 := 3;
   Program10.RopeUnit4_1 := 16#02;
   Program10.RopeUnit4_2 := 16#02;
   Program10.FilmForce4 := 30;
   Program10.FilmPrestretch4 := 200;
   Program10.Spare3H4 := 0;
   Program10.Spare64 := 0;
   Program10.Spare65 := 0;
   Program10.Spare66 := 0;
   Program10.Spare67 := 0;
   Program10.Spare68 := 0;
   Program10.Overlap4_5 := 0;
   Program10.Height5 := 50;
   Program10.Landmark5 := FALSE;
   Program10.Lifter5 := FALSE;
   Program10.SpareBit1H5 := FALSE;
   Program10.Airblower5 := TRUE;
   Program10.NextStep5 := FALSE;
   Program10.PressureP5 := FALSE;
   Program10.SpareByte2H5 := 16#00;
   Program10.Revolution5 := 1;
   Program10.RopeUnit5_1 := 16#01;
   Program10.RopeUnit5_2 := 16#01;
   Program10.FilmForce5 := 30;
   Program10.FilmPrestretch5 := 200;
   Program10.Spare3H5 := 0;
   Program10.Spare69 := 0;
   Program10.Spare70 := 0;
   Program10.Spare71 := 0;
   Program10.Spare72 := 0;
   Program10.Spare73 := 0;
   Program10.Overlap5_6 := 100;
   Program10.Height6 := 50;
   Program10.Landmark6 := FALSE;
   Program10.Lifter6 := FALSE;
   Program10.SpareBit1H6 := FALSE;
   Program10.Airblower6 := TRUE;
   Program10.NextStep6 := FALSE;
   Program10.PressureP6 := FALSE;
   Program10.SpareByte2H6 := 16#00;
   Program10.Revolution6 := 2;
   Program10.RopeUnit6_1 := 16#02;
   Program10.RopeUnit6_2 := 16#01;
   Program10.FilmForce6 := 20;
   Program10.FilmPrestretch6 := 200;
   Program10.Spare3H6 := 0;
   Program10.Spare74 := 0;
   Program10.Spare75 := 0;
   Program10.Spare76 := 0;
   Program10.Spare77 := 0;
   Program10.Spare78 := 0;
   Program10.Overlap6_7 := 0;
   Program10.Height7 := 0;
   Program10.Landmark7 := FALSE;
   Program10.Lifter7 := FALSE;
   Program10.SpareBit1H7 := FALSE;
   Program10.Airblower7 := FALSE;
   Program10.NextStep7 := TRUE;
   Program10.PressureP7 := FALSE;
   Program10.SpareByte2H7 := 16#00;
   Program10.Revolution7 := 1;
   Program10.RopeUnit7_1 := 16#01;
   Program10.RopeUnit7_2 := 16#01;
   Program10.FilmForce7 := 0;
   Program10.FilmPrestretch7 := 100;
   Program10.Spare3H7 := 0;
   Program10.Spare79 := 0;
   Program10.Spare80 := 0;
   Program10.Spare81 := 0;
   Program10.Spare82 := 0;
   Program10.Spare83 := 0;
   Program10.Overlap7_8 := 0;
   Program10.Height8 := 0;
   Program10.Landmark8 := FALSE;
   Program10.Lifter8 := FALSE;
   Program10.SpareBit1H8 := FALSE;
   Program10.Airblower8 := FALSE;
   Program10.NextStep8 := TRUE;
   Program10.PressureP8 := FALSE;
   Program10.SpareByte2H8 := 16#00;
   Program10.Revolution8 := 1;
   Program10.RopeUnit8_1 := 16#01;
   Program10.RopeUnit8_2 := 16#01;
   Program10.FilmForce8 := 0;
   Program10.FilmPrestretch8 := 100;
   Program10.Spare3H8 := 0;
   Program10.Spare84 := 0;
   Program10.Spare85 := 0;
   Program10.Spare86 := 0;
   Program10.Spare87 := 0;
   Program10.Spare88 := 0;
   Program10.Overlap8_9 := 0;
   Program10.Height9 := 0;
   Program10.Landmark9 := FALSE;
   Program10.Lifter9 := FALSE;
   Program10.SpareBit1H9 := FALSE;
   Program10.Airblower9 := FALSE;
   Program10.NextStep9 := TRUE;
   Program10.PressureP9 := FALSE;
   Program10.SpareByte2H9 := 16#00;
   Program10.Revolution9 := 1;
   Program10.RopeUnit9_1 := 16#01;
   Program10.RopeUnit9_2 := 16#01;
   Program10.FilmForce9 := 0;
   Program10.FilmPrestretch9 := 100;
   Program10.Spare3H9 := 0;
   Program10.Spare89 := 0;
   Program10.Spare90 := 0;
   Program10.Spare91 := 0;
   Program10.Spare92 := 0;
   Program10.Spare93 := 0;
   Program10.Overlap9_10 := 0;
   Program10.Height10 := 0;
   Program10.Landmark10 := FALSE;
   Program10.Lifter10 := FALSE;
   Program10.SpareBit1H10 := FALSE;
   Program10.Airblower10 := FALSE;
   Program10.NextStep10 := FALSE;
   Program10.PressureP10 := FALSE;
   Program10.SpareByte2H10 := 16#00;
   Program10.Revolution10 := 1;
   Program10.RopeUnit10_1 := 16#01;
   Program10.RopeUnit10_2 := 16#01;
   Program10.FilmForce10 := 0;
   Program10.FilmPrestretch10 := 100;
   Program10.Spare3H10 := 0;
   Program10.Spare94 := 0;
   Program10.Spare95 := 0;
   Program10.Spare96 := 0;
   Program10.Spare97 := 0;
   Program10.Spare98 := 0;
   Program10.Overlap10_11 := 0;
   Program10.Height11 := 0;
   Program10.Landmark11 := FALSE;
   Program10.Lifter11 := FALSE;
   Program10.SpareBit1H11 := FALSE;
   Program10.Airblower11 := FALSE;
   Program10.NextStep11 := TRUE;
   Program10.PressureP11 := FALSE;
   Program10.SpareByte2H11 := 16#00;
   Program10.Revolution11 := 1;
   Program10.RopeUnit11_1 := 16#01;
   Program10.RopeUnit11_2 := 16#01;
   Program10.FilmForce11 := 0;
   Program10.FilmPrestretch11 := 100;
   Program10.Spare3H11 := 0;
   Program10.Spare99 := 0;
   Program10.Spare100 := 0;
   Program10.Spare101 := 0;
   Program10.Spare102 := 0;
   Program10.Spare103 := 0;
   Program10.Overlap11_12 := 0;
   Program10.Height12 := 0;
   Program10.Landmark12 := FALSE;
   Program10.Lifter12 := FALSE;
   Program10.SpareBit1H12 := FALSE;
   Program10.Airblower12 := FALSE;
   Program10.NextStep12 := FALSE;
   Program10.PressureP12 := FALSE;
   Program10.SpareByte2H12 := 16#00;
   Program10.Revolution12 := 1;
   Program10.RopeUnit12_1 := 16#01;
   Program10.RopeUnit12_2 := 16#01;
   Program10.FilmForce12 := 0;
   Program10.FilmPrestretch12 := 100;
   Program10.Spare3H12 := 0;
   Program10.Spare104 := 0;
   Program10.Spare105 := 0;
   Program10.Spare106 := 0;
   Program10.Spare107 := 0;
   Program10.Spare108 := 0;
END_DATA_BLOCK

DATA_BLOCK "DB243_Program7"   // DB243
{ S7_Optimized_Access := 'FALSE' }
AUTHOR : Robopac
VERSION : 0.0
// stored: AutoNumber false, IsOnlyStoredInLoadMemory false, IsWriteProtectedInAS false
   VAR RETAIN
      Program7 { S7_SetPoint := 'True'} : "DatiProgramma";
   END_VAR
BEGIN
   Program7.Wrapping := TRUE;
   Program7.TopLenght := 500;
   Program7.TopRelease := 0;
   Program7.TopDown := 0;
   Program7.Top := 4;
   Program7.PressurePTime := 0;
   Program7.LifterTime := 0;
   Program7.RevOverContrast := 1;
   Program7.RopeEndCycle := 16#01;
   Program7.Spare4 := 16#01;
   Program7.RopeTime := 1500;
   Program7.RevOverClamp := 1;
   Program7.FilmForceFinalRev := 15;
   Program7.FilmPrestretchFinalRev := 100;
   Program7.ArmSpeed := 100;
   Program7.CarriageDown4Top := 500;
   Program7.TopDownTime := 1500;
   Program7.LapsUnderTop := 0;
   Program7.Spare6 := 0;
   Program7.Spare7 := 0;
   Program7.Spare8 := 0;
   Program7.Spare9 := 0;
   Program7.Spare10 := 0;
   Program7.Spare11 := 0;
   Program7.Spare12 := 0;
   Program7.Overlap0_1 := 0;
   Program7.Height1 := 15;
   Program7.Landmark1 := FALSE;
   Program7.Lifter1 := FALSE;
   Program7.SpareBit1H1 := FALSE;
   Program7.Airblower1 := TRUE;
   Program7.NextStep1 := TRUE;
   Program7.PressureP1 := TRUE;
   Program7.SpareByte2H1 := 16#00;
   Program7.Revolution1 := 0;
   Program7.RopeUnit1_1 := 16#02;
   Program7.RopeUnit1_2 := 16#01;
   Program7.FilmForce1 := 5;
   Program7.FilmPrestretch1 := 200;
   Program7.Spare3H1 := 0;
   Program7.Spare49 := 0;
   Program7.Spare50 := 0;
   Program7.Spare51 := 0;
   Program7.Spare52 := 0;
   Program7.Spare53 := 0;
   Program7.Overlap1_2 := 0;
   Program7.Height2 := 80;
   Program7.Landmark2 := FALSE;
   Program7.Lifter2 := FALSE;
   Program7.SpareBit1H2 := FALSE;
   Program7.Airblower2 := TRUE;
   Program7.NextStep2 := TRUE;
   Program7.PressureP2 := TRUE;
   Program7.SpareByte2H2 := 16#00;
   Program7.Revolution2 := 1;
   Program7.RopeUnit2_1 := 16#01;
   Program7.RopeUnit2_2 := 16#01;
   Program7.FilmForce2 := 15;
   Program7.FilmPrestretch2 := 200;
   Program7.Spare3H2 := 0;
   Program7.Spare54 := 0;
   Program7.Spare55 := 0;
   Program7.Spare56 := 0;
   Program7.Spare57 := 0;
   Program7.Spare58 := 0;
   Program7.Overlap2_3 := 0;
   Program7.Height3 := 120;
   Program7.Landmark3 := FALSE;
   Program7.Lifter3 := FALSE;
   Program7.SpareBit1H3 := FALSE;
   Program7.Airblower3 := TRUE;
   Program7.NextStep3 := TRUE;
   Program7.PressureP3 := TRUE;
   Program7.SpareByte2H3 := 16#00;
   Program7.Revolution3 := 1;
   Program7.RopeUnit3_1 := 16#01;
   Program7.RopeUnit3_2 := 16#01;
   Program7.FilmForce3 := 25;
   Program7.FilmPrestretch3 := 200;
   Program7.Spare3H3 := 0;
   Program7.Spare59 := 0;
   Program7.Spare60 := 0;
   Program7.Spare61 := 380;
   Program7.Spare62 := 2800;
   Program7.Spare63 := 0;
   Program7.Overlap3_4 := 0;
   Program7.Height4 := -100;
   Program7.Landmark4 := TRUE;
   Program7.Lifter4 := FALSE;
   Program7.SpareBit1H4 := FALSE;
   Program7.Airblower4 := FALSE;
   Program7.NextStep4 := TRUE;
   Program7.PressureP4 := TRUE;
   Program7.SpareByte2H4 := 16#00;
   Program7.Revolution4 := 1;
   Program7.RopeUnit4_1 := 16#01;
   Program7.RopeUnit4_2 := 16#01;
   Program7.FilmForce4 := 20;
   Program7.FilmPrestretch4 := 200;
   Program7.Spare3H4 := 0;
   Program7.Spare64 := 0;
   Program7.Spare65 := 0;
   Program7.Spare66 := 0;
   Program7.Spare67 := 0;
   Program7.Spare68 := 0;
   Program7.Overlap4_5 := 300;
   Program7.Height5 := 120;
   Program7.Landmark5 := FALSE;
   Program7.Lifter5 := FALSE;
   Program7.SpareBit1H5 := FALSE;
   Program7.Airblower5 := TRUE;
   Program7.NextStep5 := TRUE;
   Program7.PressureP5 := FALSE;
   Program7.SpareByte2H5 := 16#00;
   Program7.Revolution5 := 2;
   Program7.RopeUnit5_1 := 16#02;
   Program7.RopeUnit5_2 := 16#02;
   Program7.FilmForce5 := 15;
   Program7.FilmPrestretch5 := 200;
   Program7.Spare3H5 := 0;
   Program7.Spare69 := 0;
   Program7.Spare70 := 0;
   Program7.Spare71 := 0;
   Program7.Spare72 := 0;
   Program7.Spare73 := 0;
   Program7.Overlap5_6 := 300;
   Program7.Height6 := 85;
   Program7.Landmark6 := FALSE;
   Program7.Lifter6 := FALSE;
   Program7.SpareBit1H6 := FALSE;
   Program7.Airblower6 := TRUE;
   Program7.NextStep6 := FALSE;
   Program7.PressureP6 := FALSE;
   Program7.SpareByte2H6 := 16#00;
   Program7.Revolution6 := 1;
   Program7.RopeUnit6_1 := 16#01;
   Program7.RopeUnit6_2 := 16#01;
   Program7.FilmForce6 := 20;
   Program7.FilmPrestretch6 := 200;
   Program7.Spare3H6 := 0;
   Program7.Spare74 := 0;
   Program7.Spare75 := 0;
   Program7.Spare76 := 0;
   Program7.Spare77 := 0;
   Program7.Spare78 := 0;
   Program7.Overlap6_7 := 0;
   Program7.Height7 := 0;
   Program7.Landmark7 := FALSE;
   Program7.Lifter7 := FALSE;
   Program7.SpareBit1H7 := FALSE;
   Program7.Airblower7 := FALSE;
   Program7.NextStep7 := TRUE;
   Program7.PressureP7 := FALSE;
   Program7.SpareByte2H7 := 16#00;
   Program7.Revolution7 := 1;
   Program7.RopeUnit7_1 := 16#01;
   Program7.RopeUnit7_2 := 16#01;
   Program7.FilmForce7 := 0;
   Program7.FilmPrestretch7 := 100;
   Program7.Spare3H7 := 0;
   Program7.Spare79 := 0;
   Program7.Spare80 := 0;
   Program7.Spare81 := 0;
   Program7.Spare82 := 0;
   Program7.Spare83 := 0;
   Program7.Overlap7_8 := 0;
   Program7.Height8 := 0;
   Program7.Landmark8 := FALSE;
   Program7.Lifter8 := FALSE;
   Program7.SpareBit1H8 := FALSE;
   Program7.Airblower8 := FALSE;
   Program7.NextStep8 := TRUE;
   Program7.PressureP8 := FALSE;
   Program7.SpareByte2H8 := 16#00;
   Program7.Revolution8 := 1;
   Program7.RopeUnit8_1 := 16#01;
   Program7.RopeUnit8_2 := 16#01;
   Program7.FilmForce8 := 0;
   Program7.FilmPrestretch8 := 100;
   Program7.Spare3H8 := 0;
   Program7.Spare84 := 0;
   Program7.Spare85 := 0;
   Program7.Spare86 := 0;
   Program7.Spare87 := 0;
   Program7.Spare88 := 0;
   Program7.Overlap8_9 := 0;
   Program7.Height9 := 0;
   Program7.Landmark9 := FALSE;
   Program7.Lifter9 := FALSE;
   Program7.SpareBit1H9 := FALSE;
   Program7.Airblower9 := FALSE;
   Program7.NextStep9 := TRUE;
   Program7.PressureP9 := FALSE;
   Program7.SpareByte2H9 := 16#00;
   Program7.Revolution9 := 1;
   Program7.RopeUnit9_1 := 16#01;
   Program7.RopeUnit9_2 := 16#01;
   Program7.FilmForce9 := 0;
   Program7.FilmPrestretch9 := 100;
   Program7.Spare3H9 := 0;
   Program7.Spare89 := 0;
   Program7.Spare90 := 0;
   Program7.Spare91 := 0;
   Program7.Spare92 := 0;
   Program7.Spare93 := 0;
   Program7.Overlap9_10 := 0;
   Program7.Height10 := 0;
   Program7.Landmark10 := FALSE;
   Program7.Lifter10 := FALSE;
   Program7.SpareBit1H10 := FALSE;
   Program7.Airblower10 := FALSE;
   Program7.NextStep10 := FALSE;
   Program7.PressureP10 := FALSE;
   Program7.SpareByte2H10 := 16#00;
   Program7.Revolution10 := 1;
   Program7.RopeUnit10_1 := 16#01;
   Program7.RopeUnit10_2 := 16#01;
   Program7.FilmForce10 := 0;
   Program7.FilmPrestretch10 := 100;
   Program7.Spare3H10 := 0;
   Program7.Spare94 := 0;
   Program7.Spare95 := 0;
   Program7.Spare96 := 0;
   Program7.Spare97 := 0;
   Program7.Spare98 := 0;
   Program7.Overlap10_11 := 0;
   Program7.Height11 := 0;
   Program7.Landmark11 := FALSE;
   Program7.Lifter11 := FALSE;
   Program7.SpareBit1H11 := FALSE;
   Program7.Airblower11 := FALSE;
   Program7.NextStep11 := TRUE;
   Program7.PressureP11 := FALSE;
   Program7.SpareByte2H11 := 16#00;
   Program7.Revolution11 := 1;
   Program7.RopeUnit11_1 := 16#01;
   Program7.RopeUnit11_2 := 16#01;
   Program7.FilmForce11 := 0;
   Program7.FilmPrestretch11 := 100;
   Program7.Spare3H11 := 0;
   Program7.Spare99 := 0;
   Program7.Spare100 := 0;
   Program7.Spare101 := 0;
   Program7.Spare102 := 0;
   Program7.Spare103 := 0;
   Program7.Overlap11_12 := 0;
   Program7.Height12 := 0;
   Program7.Landmark12 := FALSE;
   Program7.Lifter12 := FALSE;
   Program7.SpareBit1H12 := FALSE;
   Program7.Airblower12 := FALSE;
   Program7.NextStep12 := FALSE;
   Program7.PressureP12 := FALSE;
   Program7.SpareByte2H12 := 16#00;
   Program7.Revolution12 := 1;
   Program7.RopeUnit12_1 := 16#01;
   Program7.RopeUnit12_2 := 16#01;
   Program7.FilmForce12 := 0;
   Program7.FilmPrestretch12 := 100;
   Program7.Spare3H12 := 0;
   Program7.Spare104 := 0;
   Program7.Spare105 := 0;
   Program7.Spare106 := 0;
   Program7.Spare107 := 0;
   Program7.Spare108 := 0;
END_DATA_BLOCK

DATA_BLOCK "DB246_Program4"   // DB246
{ S7_Optimized_Access := 'FALSE' }
AUTHOR : Robopac
VERSION : 0.0
// stored: AutoNumber false, IsOnlyStoredInLoadMemory false, IsWriteProtectedInAS false
   VAR RETAIN
      Program4 { S7_SetPoint := 'True'} : "DatiProgramma";
   END_VAR
BEGIN
   Program4.Wrapping := TRUE;
   Program4.TopLenght := 500;
   Program4.TopRelease := 0;
   Program4.TopDown := 0;
   Program4.Top := 4;
   Program4.PressurePTime := 0;
   Program4.LifterTime := 0;
   Program4.RevOverContrast := 1;
   Program4.RopeEndCycle := 16#02;
   Program4.Spare4 := 16#01;
   Program4.RopeTime := 1500;
   Program4.RevOverClamp := 1;
   Program4.FilmForceFinalRev := 10;
   Program4.FilmPrestretchFinalRev := 100;
   Program4.ArmSpeed := 100;
   Program4.CarriageDown4Top := 500;
   Program4.TopDownTime := 1500;
   Program4.LapsUnderTop := 0;
   Program4.Spare6 := 0;
   Program4.Spare7 := 0;
   Program4.Spare8 := 0;
   Program4.Spare9 := 0;
   Program4.Spare10 := 0;
   Program4.Spare11 := 0;
   Program4.Spare12 := 0;
   Program4.Overlap0_1 := 0;
   Program4.Height1 := 130;
   Program4.Landmark1 := FALSE;
   Program4.Lifter1 := FALSE;
   Program4.SpareBit1H1 := FALSE;
   Program4.Airblower1 := TRUE;
   Program4.NextStep1 := TRUE;
   Program4.PressureP1 := TRUE;
   Program4.SpareByte2H1 := 16#00;
   Program4.Revolution1 := 1;
   Program4.RopeUnit1_1 := 16#01;
   Program4.RopeUnit1_2 := 16#01;
   Program4.FilmForce1 := 5;
   Program4.FilmPrestretch1 := 200;
   Program4.Spare3H1 := 0;
   Program4.Spare49 := 0;
   Program4.Spare50 := 0;
   Program4.Spare51 := 0;
   Program4.Spare52 := 0;
   Program4.Spare53 := 0;
   Program4.Overlap1_2 := 0;
   Program4.Height2 := 50;
   Program4.Landmark2 := FALSE;
   Program4.Lifter2 := FALSE;
   Program4.SpareBit1H2 := FALSE;
   Program4.Airblower2 := TRUE;
   Program4.NextStep2 := TRUE;
   Program4.PressureP2 := TRUE;
   Program4.SpareByte2H2 := 16#00;
   Program4.Revolution2 := 1;
   Program4.RopeUnit2_1 := 16#01;
   Program4.RopeUnit2_2 := 16#01;
   Program4.FilmForce2 := 20;
   Program4.FilmPrestretch2 := 200;
   Program4.Spare3H2 := 0;
   Program4.Spare54 := 0;
   Program4.Spare55 := 0;
   Program4.Spare56 := 0;
   Program4.Spare57 := 0;
   Program4.Spare58 := 0;
   Program4.Overlap2_3 := 100;
   Program4.Height3 := -50;
   Program4.Landmark3 := TRUE;
   Program4.Lifter3 := FALSE;
   Program4.SpareBit1H3 := FALSE;
   Program4.Airblower3 := TRUE;
   Program4.NextStep3 := TRUE;
   Program4.PressureP3 := TRUE;
   Program4.SpareByte2H3 := 16#00;
   Program4.Revolution3 := 2;
   Program4.RopeUnit3_1 := 16#01;
   Program4.RopeUnit3_2 := 16#01;
   Program4.FilmForce3 := 30;
   Program4.FilmPrestretch3 := 200;
   Program4.Spare3H3 := 0;
   Program4.Spare59 := 0;
   Program4.Spare60 := 0;
   Program4.Spare61 := 380;
   Program4.Spare62 := 2800;
   Program4.Spare63 := 0;
   Program4.Overlap3_4 := 100;
   Program4.Height4 := 100;
   Program4.Landmark4 := FALSE;
   Program4.Lifter4 := FALSE;
   Program4.SpareBit1H4 := FALSE;
   Program4.Airblower4 := TRUE;
   Program4.NextStep4 := TRUE;
   Program4.PressureP4 := TRUE;
   Program4.SpareByte2H4 := 16#00;
   Program4.Revolution4 := 3;
   Program4.RopeUnit4_1 := 16#02;
   Program4.RopeUnit4_2 := 16#02;
   Program4.FilmForce4 := 30;
   Program4.FilmPrestretch4 := 200;
   Program4.Spare3H4 := 0;
   Program4.Spare64 := 0;
   Program4.Spare65 := 0;
   Program4.Spare66 := 0;
   Program4.Spare67 := 0;
   Program4.Spare68 := 0;
   Program4.Overlap4_5 := 0;
   Program4.Height5 := 50;
   Program4.Landmark5 := FALSE;
   Program4.Lifter5 := FALSE;
   Program4.SpareBit1H5 := FALSE;
   Program4.Airblower5 := TRUE;
   Program4.NextStep5 := FALSE;
   Program4.PressureP5 := FALSE;
   Program4.SpareByte2H5 := 16#00;
   Program4.Revolution5 := 1;
   Program4.RopeUnit5_1 := 16#01;
   Program4.RopeUnit5_2 := 16#01;
   Program4.FilmForce5 := 30;
   Program4.FilmPrestretch5 := 200;
   Program4.Spare3H5 := 0;
   Program4.Spare69 := 0;
   Program4.Spare70 := 0;
   Program4.Spare71 := 0;
   Program4.Spare72 := 0;
   Program4.Spare73 := 0;
   Program4.Overlap5_6 := 100;
   Program4.Height6 := 50;
   Program4.Landmark6 := FALSE;
   Program4.Lifter6 := FALSE;
   Program4.SpareBit1H6 := FALSE;
   Program4.Airblower6 := TRUE;
   Program4.NextStep6 := FALSE;
   Program4.PressureP6 := FALSE;
   Program4.SpareByte2H6 := 16#00;
   Program4.Revolution6 := 2;
   Program4.RopeUnit6_1 := 16#02;
   Program4.RopeUnit6_2 := 16#01;
   Program4.FilmForce6 := 20;
   Program4.FilmPrestretch6 := 200;
   Program4.Spare3H6 := 0;
   Program4.Spare74 := 0;
   Program4.Spare75 := 0;
   Program4.Spare76 := 0;
   Program4.Spare77 := 0;
   Program4.Spare78 := 0;
   Program4.Overlap6_7 := 0;
   Program4.Height7 := 0;
   Program4.Landmark7 := FALSE;
   Program4.Lifter7 := FALSE;
   Program4.SpareBit1H7 := FALSE;
   Program4.Airblower7 := FALSE;
   Program4.NextStep7 := TRUE;
   Program4.PressureP7 := FALSE;
   Program4.SpareByte2H7 := 16#00;
   Program4.Revolution7 := 1;
   Program4.RopeUnit7_1 := 16#01;
   Program4.RopeUnit7_2 := 16#01;
   Program4.FilmForce7 := 0;
   Program4.FilmPrestretch7 := 100;
   Program4.Spare3H7 := 0;
   Program4.Spare79 := 0;
   Program4.Spare80 := 0;
   Program4.Spare81 := 0;
   Program4.Spare82 := 0;
   Program4.Spare83 := 0;
   Program4.Overlap7_8 := 0;
   Program4.Height8 := 0;
   Program4.Landmark8 := FALSE;
   Program4.Lifter8 := FALSE;
   Program4.SpareBit1H8 := FALSE;
   Program4.Airblower8 := FALSE;
   Program4.NextStep8 := TRUE;
   Program4.PressureP8 := FALSE;
   Program4.SpareByte2H8 := 16#00;
   Program4.Revolution8 := 1;
   Program4.RopeUnit8_1 := 16#01;
   Program4.RopeUnit8_2 := 16#01;
   Program4.FilmForce8 := 0;
   Program4.FilmPrestretch8 := 100;
   Program4.Spare3H8 := 0;
   Program4.Spare84 := 0;
   Program4.Spare85 := 0;
   Program4.Spare86 := 0;
   Program4.Spare87 := 0;
   Program4.Spare88 := 0;
   Program4.Overlap8_9 := 0;
   Program4.Height9 := 0;
   Program4.Landmark9 := FALSE;
   Program4.Lifter9 := FALSE;
   Program4.SpareBit1H9 := FALSE;
   Program4.Airblower9 := FALSE;
   Program4.NextStep9 := TRUE;
   Program4.PressureP9 := FALSE;
   Program4.SpareByte2H9 := 16#00;
   Program4.Revolution9 := 1;
   Program4.RopeUnit9_1 := 16#01;
   Program4.RopeUnit9_2 := 16#01;
   Program4.FilmForce9 := 0;
   Program4.FilmPrestretch9 := 100;
   Program4.Spare3H9 := 0;
   Program4.Spare89 := 0;
   Program4.Spare90 := 0;
   Program4.Spare91 := 0;
   Program4.Spare92 := 0;
   Program4.Spare93 := 0;
   Program4.Overlap9_10 := 0;
   Program4.Height10 := 0;
   Program4.Landmark10 := FALSE;
   Program4.Lifter10 := FALSE;
   Program4.SpareBit1H10 := FALSE;
   Program4.Airblower10 := FALSE;
   Program4.NextStep10 := FALSE;
   Program4.PressureP10 := FALSE;
   Program4.SpareByte2H10 := 16#00;
   Program4.Revolution10 := 1;
   Program4.RopeUnit10_1 := 16#01;
   Program4.RopeUnit10_2 := 16#01;
   Program4.FilmForce10 := 0;
   Program4.FilmPrestretch10 := 100;
   Program4.Spare3H10 := 0;
   Program4.Spare94 := 0;
   Program4.Spare95 := 0;
   Program4.Spare96 := 0;
   Program4.Spare97 := 0;
   Program4.Spare98 := 0;
   Program4.Overlap10_11 := 0;
   Program4.Height11 := 0;
   Program4.Landmark11 := FALSE;
   Program4.Lifter11 := FALSE;
   Program4.SpareBit1H11 := FALSE;
   Program4.Airblower11 := FALSE;
   Program4.NextStep11 := TRUE;
   Program4.PressureP11 := FALSE;
   Program4.SpareByte2H11 := 16#00;
   Program4.Revolution11 := 1;
   Program4.RopeUnit11_1 := 16#01;
   Program4.RopeUnit11_2 := 16#01;
   Program4.FilmForce11 := 0;
   Program4.FilmPrestretch11 := 100;
   Program4.Spare3H11 := 0;
   Program4.Spare99 := 0;
   Program4.Spare100 := 0;
   Program4.Spare101 := 0;
   Program4.Spare102 := 0;
   Program4.Spare103 := 0;
   Program4.Overlap11_12 := 0;
   Program4.Height12 := 0;
   Program4.Landmark12 := FALSE;
   Program4.Lifter12 := FALSE;
   Program4.SpareBit1H12 := FALSE;
   Program4.Airblower12 := FALSE;
   Program4.NextStep12 := FALSE;
   Program4.PressureP12 := FALSE;
   Program4.SpareByte2H12 := 16#00;
   Program4.Revolution12 := 1;
   Program4.RopeUnit12_1 := 16#01;
   Program4.RopeUnit12_2 := 16#01;
   Program4.FilmForce12 := 0;
   Program4.FilmPrestretch12 := 100;
   Program4.Spare3H12 := 0;
   Program4.Spare104 := 0;
   Program4.Spare105 := 0;
   Program4.Spare106 := 0;
   Program4.Spare107 := 0;
   Program4.Spare108 := 0;
END_DATA_BLOCK

DATA_BLOCK "DB249_Program1"   // DB249
{ S7_Optimized_Access := 'FALSE' }
AUTHOR : Robopac
VERSION : 0.0
// stored: AutoNumber false, IsOnlyStoredInLoadMemory false, IsWriteProtectedInAS false
   VAR RETAIN
      Program1 { S7_SetPoint := 'True'} : "DatiProgramma";
   END_VAR
BEGIN
   Program1.Wrapping := TRUE;
   Program1.TopLenght := 500;
   Program1.TopRelease := 0;
   Program1.TopDown := 0;
   Program1.Top := 4;
   Program1.PressurePTime := 0;
   Program1.LifterTime := 0;
   Program1.RevOverContrast := 1;
   Program1.RopeEndCycle := 16#02;
   Program1.Spare4 := 16#01;
   Program1.RopeTime := 1500;
   Program1.RevOverClamp := 1;
   Program1.FilmForceFinalRev := 25;
   Program1.FilmPrestretchFinalRev := 100;
   Program1.ArmSpeed := 87;
   Program1.CarriageDown4Top := 500;
   Program1.TopDownTime := 1500;
   Program1.LapsUnderTop := 0;
   Program1.Spare6 := 0;
   Program1.Spare7 := 0;
   Program1.Spare8 := 0;
   Program1.Spare9 := 0;
   Program1.Spare10 := 0;
   Program1.Spare11 := 0;
   Program1.Spare12 := 0;
   Program1.Overlap0_1 := 0;
   Program1.Height1 := 120;
   Program1.Landmark1 := FALSE;
   Program1.Lifter1 := FALSE;
   Program1.SpareBit1H1 := FALSE;
   Program1.Airblower1 := TRUE;
   Program1.NextStep1 := TRUE;
   Program1.PressureP1 := TRUE;
   Program1.SpareByte2H1 := 16#00;
   Program1.Revolution1 := 1;
   Program1.RopeUnit1_1 := 16#03;
   Program1.RopeUnit1_2 := 16#01;
   Program1.FilmForce1 := 5;
   Program1.FilmPrestretch1 := 200;
   Program1.Spare3H1 := 0;
   Program1.Spare49 := 0;
   Program1.Spare50 := 0;
   Program1.Spare51 := 0;
   Program1.Spare52 := 0;
   Program1.Spare53 := 0;
   Program1.Overlap1_2 := 0;
   Program1.Height2 := 85;
   Program1.Landmark2 := FALSE;
   Program1.Lifter2 := FALSE;
   Program1.SpareBit1H2 := FALSE;
   Program1.Airblower2 := TRUE;
   Program1.NextStep2 := TRUE;
   Program1.PressureP2 := TRUE;
   Program1.SpareByte2H2 := 16#00;
   Program1.Revolution2 := 3;
   Program1.RopeUnit2_1 := 16#01;
   Program1.RopeUnit2_2 := 16#01;
   Program1.FilmForce2 := 15;
   Program1.FilmPrestretch2 := 200;
   Program1.Spare3H2 := 0;
   Program1.Spare54 := 0;
   Program1.Spare55 := 0;
   Program1.Spare56 := 0;
   Program1.Spare57 := 0;
   Program1.Spare58 := 0;
   Program1.Overlap2_3 := 300;
   Program1.Height3 := 110;
   Program1.Landmark3 := FALSE;
   Program1.Lifter3 := FALSE;
   Program1.SpareBit1H3 := FALSE;
   Program1.Airblower3 := TRUE;
   Program1.NextStep3 := TRUE;
   Program1.PressureP3 := TRUE;
   Program1.SpareByte2H3 := 16#00;
   Program1.Revolution3 := 2;
   Program1.RopeUnit3_1 := 16#03;
   Program1.RopeUnit3_2 := 16#03;
   Program1.FilmForce3 := 20;
   Program1.FilmPrestretch3 := 200;
   Program1.Spare3H3 := 0;
   Program1.Spare59 := 0;
   Program1.Spare60 := 0;
   Program1.Spare61 := 380;
   Program1.Spare62 := 2800;
   Program1.Spare63 := 0;
   Program1.Overlap3_4 := 100;
   Program1.Height4 := -100;
   Program1.Landmark4 := TRUE;
   Program1.Lifter4 := FALSE;
   Program1.SpareBit1H4 := FALSE;
   Program1.Airblower4 := FALSE;
   Program1.NextStep4 := TRUE;
   Program1.PressureP4 := TRUE;
   Program1.SpareByte2H4 := 16#00;
   Program1.Revolution4 := 1;
   Program1.RopeUnit4_1 := 16#01;
   Program1.RopeUnit4_2 := 16#01;
   Program1.FilmForce4 := 18;
   Program1.FilmPrestretch4 := 200;
   Program1.Spare3H4 := 0;
   Program1.Spare64 := 0;
   Program1.Spare65 := 0;
   Program1.Spare66 := 0;
   Program1.Spare67 := 0;
   Program1.Spare68 := 0;
   Program1.Overlap4_5 := 100;
   Program1.Height5 := 60;
   Program1.Landmark5 := FALSE;
   Program1.Lifter5 := FALSE;
   Program1.SpareBit1H5 := FALSE;
   Program1.Airblower5 := TRUE;
   Program1.NextStep5 := TRUE;
   Program1.PressureP5 := FALSE;
   Program1.SpareByte2H5 := 16#00;
   Program1.Revolution5 := 1;
   Program1.RopeUnit5_1 := 16#01;
   Program1.RopeUnit5_2 := 16#01;
   Program1.FilmForce5 := 25;
   Program1.FilmPrestretch5 := 200;
   Program1.Spare3H5 := 0;
   Program1.Spare69 := 0;
   Program1.Spare70 := 0;
   Program1.Spare71 := 0;
   Program1.Spare72 := 0;
   Program1.Spare73 := 0;
   Program1.Overlap5_6 := 100;
   Program1.Height6 := 40;
   Program1.Landmark6 := FALSE;
   Program1.Lifter6 := FALSE;
   Program1.SpareBit1H6 := FALSE;
   Program1.Airblower6 := TRUE;
   Program1.NextStep6 := FALSE;
   Program1.PressureP6 := FALSE;
   Program1.SpareByte2H6 := 16#00;
   Program1.Revolution6 := 1;
   Program1.RopeUnit6_1 := 16#01;
   Program1.RopeUnit6_2 := 16#01;
   Program1.FilmForce6 := 15;
   Program1.FilmPrestretch6 := 200;
   Program1.Spare3H6 := 0;
   Program1.Spare74 := 0;
   Program1.Spare75 := 0;
   Program1.Spare76 := 0;
   Program1.Spare77 := 0;
   Program1.Spare78 := 0;
   Program1.Overlap6_7 := 0;
   Program1.Height7 := 0;
   Program1.Landmark7 := FALSE;
   Program1.Lifter7 := FALSE;
   Program1.SpareBit1H7 := FALSE;
   Program1.Airblower7 := FALSE;
   Program1.NextStep7 := TRUE;
   Program1.PressureP7 := FALSE;
   Program1.SpareByte2H7 := 16#00;
   Program1.Revolution7 := 1;
   Program1.RopeUnit7_1 := 16#01;
   Program1.RopeUnit7_2 := 16#01;
   Program1.FilmForce7 := 0;
   Program1.FilmPrestretch7 := 100;
   Program1.Spare3H7 := 0;
   Program1.Spare79 := 0;
   Program1.Spare80 := 0;
   Program1.Spare81 := 0;
   Program1.Spare82 := 0;
   Program1.Spare83 := 0;
   Program1.Overlap7_8 := 0;
   Program1.Height8 := 0;
   Program1.Landmark8 := FALSE;
   Program1.Lifter8 := FALSE;
   Program1.SpareBit1H8 := FALSE;
   Program1.Airblower8 := FALSE;
   Program1.NextStep8 := TRUE;
   Program1.PressureP8 := FALSE;
   Program1.SpareByte2H8 := 16#00;
   Program1.Revolution8 := 1;
   Program1.RopeUnit8_1 := 16#01;
   Program1.RopeUnit8_2 := 16#01;
   Program1.FilmForce8 := 0;
   Program1.FilmPrestretch8 := 100;
   Program1.Spare3H8 := 0;
   Program1.Spare84 := 0;
   Program1.Spare85 := 0;
   Program1.Spare86 := 0;
   Program1.Spare87 := 0;
   Program1.Spare88 := 0;
   Program1.Overlap8_9 := 0;
   Program1.Height9 := 0;
   Program1.Landmark9 := FALSE;
   Program1.Lifter9 := FALSE;
   Program1.SpareBit1H9 := FALSE;
   Program1.Airblower9 := FALSE;
   Program1.NextStep9 := TRUE;
   Program1.PressureP9 := FALSE;
   Program1.SpareByte2H9 := 16#00;
   Program1.Revolution9 := 1;
   Program1.RopeUnit9_1 := 16#01;
   Program1.RopeUnit9_2 := 16#01;
   Program1.FilmForce9 := 0;
   Program1.FilmPrestretch9 := 100;
   Program1.Spare3H9 := 0;
   Program1.Spare89 := 0;
   Program1.Spare90 := 0;
   Program1.Spare91 := 0;
   Program1.Spare92 := 0;
   Program1.Spare93 := 0;
   Program1.Overlap9_10 := 0;
   Program1.Height10 := 0;
   Program1.Landmark10 := FALSE;
   Program1.Lifter10 := FALSE;
   Program1.SpareBit1H10 := FALSE;
   Program1.Airblower10 := FALSE;
   Program1.NextStep10 := FALSE;
   Program1.PressureP10 := FALSE;
   Program1.SpareByte2H10 := 16#00;
   Program1.Revolution10 := 1;
   Program1.RopeUnit10_1 := 16#01;
   Program1.RopeUnit10_2 := 16#01;
   Program1.FilmForce10 := 0;
   Program1.FilmPrestretch10 := 100;
   Program1.Spare3H10 := 0;
   Program1.Spare94 := 0;
   Program1.Spare95 := 0;
   Program1.Spare96 := 0;
   Program1.Spare97 := 0;
   Program1.Spare98 := 0;
   Program1.Overlap10_11 := 0;
   Program1.Height11 := 0;
   Program1.Landmark11 := FALSE;
   Program1.Lifter11 := FALSE;
   Program1.SpareBit1H11 := FALSE;
   Program1.Airblower11 := FALSE;
   Program1.NextStep11 := TRUE;
   Program1.PressureP11 := FALSE;
   Program1.SpareByte2H11 := 16#00;
   Program1.Revolution11 := 1;
   Program1.RopeUnit11_1 := 16#01;
   Program1.RopeUnit11_2 := 16#01;
   Program1.FilmForce11 := 0;
   Program1.FilmPrestretch11 := 100;
   Program1.Spare3H11 := 0;
   Program1.Spare99 := 0;
   Program1.Spare100 := 0;
   Program1.Spare101 := 0;
   Program1.Spare102 := 0;
   Program1.Spare103 := 0;
   Program1.Overlap11_12 := 0;
   Program1.Height12 := 0;
   Program1.Landmark12 := FALSE;
   Program1.Lifter12 := FALSE;
   Program1.SpareBit1H12 := FALSE;
   Program1.Airblower12 := FALSE;
   Program1.NextStep12 := FALSE;
   Program1.PressureP12 := FALSE;
   Program1.SpareByte2H12 := 16#00;
   Program1.Revolution12 := 1;
   Program1.RopeUnit12_1 := 16#01;
   Program1.RopeUnit12_2 := 16#01;
   Program1.FilmForce12 := 0;
   Program1.FilmPrestretch12 := 100;
   Program1.Spare3H12 := 0;
   Program1.Spare104 := 0;
   Program1.Spare105 := 0;
   Program1.Spare106 := 0;
   Program1.Spare107 := 0;
   Program1.Spare108 := 0;
END_DATA_BLOCK

DATA_BLOCK "DB250_ProgramData"   // DB250
{ S7_Optimized_Access := 'FALSE' }
AUTHOR : Robopac
VERSION : 0.0
// stored: AutoNumber false, IsOnlyStoredInLoadMemory false, IsWriteProtectedInAS false
   VAR RETAIN
      Program { S7_SetPoint := 'True'} : "DatiProgramma";
   END_VAR
BEGIN
   Program.Wrapping := TRUE;
   Program.TopLenght := 500;
   Program.TopRelease := 0;
   Program.TopDown := 0;
   Program.Top := 4;
   Program.PressurePTime := 0;
   Program.LifterTime := 0;
   Program.RevOverContrast := 1;
   Program.RopeEndCycle := 16#02;
   Program.Spare4 := 16#01;
   Program.RopeTime := 1500;
   Program.RevOverClamp := 1;
   Program.FilmForceFinalRev := 10;
   Program.FilmPrestretchFinalRev := 100;
   Program.ArmSpeed := 100;
   Program.CarriageDown4Top := 500;
   Program.TopDownTime := 1500;
   Program.LapsUnderTop := 0;
   Program.Spare6 := 0;
   Program.Spare7 := 0;
   Program.Spare8 := 0;
   Program.Spare9 := 0;
   Program.Spare10 := 0;
   Program.Spare11 := 0;
   Program.Spare12 := 0;
   Program.Overlap0_1 := 0;
   Program.Height1 := 130;
   Program.Landmark1 := FALSE;
   Program.Lifter1 := FALSE;
   Program.SpareBit1H1 := FALSE;
   Program.Airblower1 := TRUE;
   Program.NextStep1 := TRUE;
   Program.PressureP1 := TRUE;
   Program.SpareByte2H1 := 16#00;
   Program.Revolution1 := 1;
   Program.RopeUnit1_1 := 16#01;
   Program.RopeUnit1_2 := 16#01;
   Program.FilmForce1 := 5;
   Program.FilmPrestretch1 := 200;
   Program.Spare3H1 := 0;
   Program.Spare49 := 0;
   Program.Spare50 := 0;
   Program.Spare51 := 0;
   Program.Spare52 := 0;
   Program.Spare53 := 0;
   Program.Overlap1_2 := 0;
   Program.Height2 := 50;
   Program.Landmark2 := FALSE;
   Program.Lifter2 := FALSE;
   Program.SpareBit1H2 := FALSE;
   Program.Airblower2 := TRUE;
   Program.NextStep2 := TRUE;
   Program.PressureP2 := TRUE;
   Program.SpareByte2H2 := 16#00;
   Program.Revolution2 := 1;
   Program.RopeUnit2_1 := 16#01;
   Program.RopeUnit2_2 := 16#01;
   Program.FilmForce2 := 20;
   Program.FilmPrestretch2 := 200;
   Program.Spare3H2 := 0;
   Program.Spare54 := 0;
   Program.Spare55 := 0;
   Program.Spare56 := 0;
   Program.Spare57 := 0;
   Program.Spare58 := 0;
   Program.Overlap2_3 := 100;
   Program.Height3 := -50;
   Program.Landmark3 := TRUE;
   Program.Lifter3 := FALSE;
   Program.SpareBit1H3 := FALSE;
   Program.Airblower3 := TRUE;
   Program.NextStep3 := TRUE;
   Program.PressureP3 := TRUE;
   Program.SpareByte2H3 := 16#00;
   Program.Revolution3 := 2;
   Program.RopeUnit3_1 := 16#01;
   Program.RopeUnit3_2 := 16#01;
   Program.FilmForce3 := 30;
   Program.FilmPrestretch3 := 200;
   Program.Spare3H3 := 0;
   Program.Spare59 := 0;
   Program.Spare60 := 0;
   Program.Spare61 := 380;
   Program.Spare62 := 2800;
   Program.Spare63 := 0;
   Program.Overlap3_4 := 100;
   Program.Height4 := 100;
   Program.Landmark4 := FALSE;
   Program.Lifter4 := FALSE;
   Program.SpareBit1H4 := FALSE;
   Program.Airblower4 := TRUE;
   Program.NextStep4 := TRUE;
   Program.PressureP4 := TRUE;
   Program.SpareByte2H4 := 16#00;
   Program.Revolution4 := 3;
   Program.RopeUnit4_1 := 16#02;
   Program.RopeUnit4_2 := 16#02;
   Program.FilmForce4 := 30;
   Program.FilmPrestretch4 := 200;
   Program.Spare3H4 := 0;
   Program.Spare64 := 0;
   Program.Spare65 := 0;
   Program.Spare66 := 0;
   Program.Spare67 := 0;
   Program.Spare68 := 0;
   Program.Overlap4_5 := 0;
   Program.Height5 := 50;
   Program.Landmark5 := FALSE;
   Program.Lifter5 := FALSE;
   Program.SpareBit1H5 := FALSE;
   Program.Airblower5 := TRUE;
   Program.NextStep5 := FALSE;
   Program.PressureP5 := FALSE;
   Program.SpareByte2H5 := 16#00;
   Program.Revolution5 := 1;
   Program.RopeUnit5_1 := 16#01;
   Program.RopeUnit5_2 := 16#01;
   Program.FilmForce5 := 30;
   Program.FilmPrestretch5 := 200;
   Program.Spare3H5 := 0;
   Program.Spare69 := 0;
   Program.Spare70 := 0;
   Program.Spare71 := 0;
   Program.Spare72 := 0;
   Program.Spare73 := 0;
   Program.Overlap5_6 := 100;
   Program.Height6 := 50;
   Program.Landmark6 := FALSE;
   Program.Lifter6 := FALSE;
   Program.SpareBit1H6 := FALSE;
   Program.Airblower6 := TRUE;
   Program.NextStep6 := FALSE;
   Program.PressureP6 := FALSE;
   Program.SpareByte2H6 := 16#00;
   Program.Revolution6 := 2;
   Program.RopeUnit6_1 := 16#02;
   Program.RopeUnit6_2 := 16#01;
   Program.FilmForce6 := 20;
   Program.FilmPrestretch6 := 200;
   Program.Spare3H6 := 0;
   Program.Spare74 := 0;
   Program.Spare75 := 0;
   Program.Spare76 := 0;
   Program.Spare77 := 0;
   Program.Spare78 := 0;
   Program.Overlap6_7 := 0;
   Program.Height7 := 0;
   Program.Landmark7 := FALSE;
   Program.Lifter7 := FALSE;
   Program.SpareBit1H7 := FALSE;
   Program.Airblower7 := FALSE;
   Program.NextStep7 := TRUE;
   Program.PressureP7 := FALSE;
   Program.SpareByte2H7 := 16#00;
   Program.Revolution7 := 1;
   Program.RopeUnit7_1 := 16#01;
   Program.RopeUnit7_2 := 16#01;
   Program.FilmForce7 := 0;
   Program.FilmPrestretch7 := 100;
   Program.Spare3H7 := 0;
   Program.Spare79 := 0;
   Program.Spare80 := 0;
   Program.Spare81 := 0;
   Program.Spare82 := 0;
   Program.Spare83 := 0;
   Program.Overlap7_8 := 0;
   Program.Height8 := 0;
   Program.Landmark8 := FALSE;
   Program.Lifter8 := FALSE;
   Program.SpareBit1H8 := FALSE;
   Program.Airblower8 := FALSE;
   Program.NextStep8 := TRUE;
   Program.PressureP8 := FALSE;
   Program.SpareByte2H8 := 16#00;
   Program.Revolution8 := 1;
   Program.RopeUnit8_1 := 16#01;
   Program.RopeUnit8_2 := 16#01;
   Program.FilmForce8 := 0;
   Program.FilmPrestretch8 := 100;
   Program.Spare3H8 := 0;
   Program.Spare84 := 0;
   Program.Spare85 := 0;
   Program.Spare86 := 0;
   Program.Spare87 := 0;
   Program.Spare88 := 0;
   Program.Overlap8_9 := 0;
   Program.Height9 := 0;
   Program.Landmark9 := FALSE;
   Program.Lifter9 := FALSE;
   Program.SpareBit1H9 := FALSE;
   Program.Airblower9 := FALSE;
   Program.NextStep9 := TRUE;
   Program.PressureP9 := FALSE;
   Program.SpareByte2H9 := 16#00;
   Program.Revolution9 := 1;
   Program.RopeUnit9_1 := 16#01;
   Program.RopeUnit9_2 := 16#01;
   Program.FilmForce9 := 0;
   Program.FilmPrestretch9 := 100;
   Program.Spare3H9 := 0;
   Program.Spare89 := 0;
   Program.Spare90 := 0;
   Program.Spare91 := 0;
   Program.Spare92 := 0;
   Program.Spare93 := 0;
   Program.Overlap9_10 := 0;
   Program.Height10 := 0;
   Program.Landmark10 := FALSE;
   Program.Lifter10 := FALSE;
   Program.SpareBit1H10 := FALSE;
   Program.Airblower10 := FALSE;
   Program.NextStep10 := FALSE;
   Program.PressureP10 := FALSE;
   Program.SpareByte2H10 := 16#00;
   Program.Revolution10 := 1;
   Program.RopeUnit10_1 := 16#01;
   Program.RopeUnit10_2 := 16#01;
   Program.FilmForce10 := 0;
   Program.FilmPrestretch10 := 100;
   Program.Spare3H10 := 0;
   Program.Spare94 := 0;
   Program.Spare95 := 0;
   Program.Spare96 := 0;
   Program.Spare97 := 0;
   Program.Spare98 := 0;
   Program.Overlap10_11 := 0;
   Program.Height11 := 0;
   Program.Landmark11 := FALSE;
   Program.Lifter11 := FALSE;
   Program.SpareBit1H11 := FALSE;
   Program.Airblower11 := FALSE;
   Program.NextStep11 := TRUE;
   Program.PressureP11 := FALSE;
   Program.SpareByte2H11 := 16#00;
   Program.Revolution11 := 1;
   Program.RopeUnit11_1 := 16#01;
   Program.RopeUnit11_2 := 16#01;
   Program.FilmForce11 := 0;
   Program.FilmPrestretch11 := 100;
   Program.Spare3H11 := 0;
   Program.Spare99 := 0;
   Program.Spare100 := 0;
   Program.Spare101 := 0;
   Program.Spare102 := 0;
   Program.Spare103 := 0;
   Program.Overlap11_12 := 0;
   Program.Height12 := 0;
   Program.Landmark12 := FALSE;
   Program.Lifter12 := FALSE;
   Program.SpareBit1H12 := FALSE;
   Program.Airblower12 := FALSE;
   Program.NextStep12 := FALSE;
   Program.PressureP12 := FALSE;
   Program.SpareByte2H12 := 16#00;
   Program.Revolution12 := 1;
   Program.RopeUnit12_1 := 16#01;
   Program.RopeUnit12_2 := 16#01;
   Program.FilmForce12 := 0;
   Program.FilmPrestretch12 := 100;
   Program.Spare3H12 := 0;
   Program.Spare104 := 0;
   Program.Spare105 := 0;
   Program.Spare106 := 0;
   Program.Spare107 := 0;
   Program.Spare108 := 0;
END_DATA_BLOCK

DATA_BLOCK "DB251_ProgramDisplay"   // DB251
{ S7_Optimized_Access := 'FALSE' }
VERSION : 0.0
// stored: AutoNumber false, IsOnlyStoredInLoadMemory false, IsWriteProtectedInAS false
   VAR RETAIN
      Display { S7_SetPoint := 'True'} : "DatiProgramma";
   END_VAR
BEGIN
   Display.Wrapping := TRUE;
   Display.TopLenght := 500;
   Display.TopRelease := 0;
   Display.TopDown := 0;
   Display.Top := 4;
   Display.PressurePTime := 0;
   Display.LifterTime := 0;
   Display.RevOverContrast := 1;
   Display.RopeEndCycle := 16#02;
   Display.Spare4 := 16#01;
   Display.RopeTime := 1500;
   Display.RevOverClamp := 1;
   Display.FilmForceFinalRev := 10;
   Display.FilmPrestretchFinalRev := 100;
   Display.ArmSpeed := 100;
   Display.CarriageDown4Top := 500;
   Display.TopDownTime := 1500;
   Display.LapsUnderTop := 0;
   Display.Spare6 := 0;
   Display.Spare7 := 0;
   Display.Spare8 := 0;
   Display.Spare9 := 0;
   Display.Spare10 := 0;
   Display.Spare11 := 0;
   Display.Spare12 := 0;
   Display.Overlap0_1 := 0;
   Display.Height1 := 130;
   Display.Landmark1 := FALSE;
   Display.Lifter1 := FALSE;
   Display.SpareBit1H1 := FALSE;
   Display.Airblower1 := TRUE;
   Display.NextStep1 := TRUE;
   Display.PressureP1 := TRUE;
   Display.SpareByte2H1 := 16#00;
   Display.Revolution1 := 1;
   Display.RopeUnit1_1 := 16#01;
   Display.RopeUnit1_2 := 16#01;
   Display.FilmForce1 := 5;
   Display.FilmPrestretch1 := 200;
   Display.Spare3H1 := 0;
   Display.Spare49 := 0;
   Display.Spare50 := 0;
   Display.Spare51 := 0;
   Display.Spare52 := 0;
   Display.Spare53 := 0;
   Display.Overlap1_2 := 0;
   Display.Height2 := 50;
   Display.Landmark2 := FALSE;
   Display.Lifter2 := FALSE;
   Display.SpareBit1H2 := FALSE;
   Display.Airblower2 := TRUE;
   Display.NextStep2 := TRUE;
   Display.PressureP2 := TRUE;
   Display.SpareByte2H2 := 16#00;
   Display.Revolution2 := 1;
   Display.RopeUnit2_1 := 16#01;
   Display.RopeUnit2_2 := 16#01;
   Display.FilmForce2 := 20;
   Display.FilmPrestretch2 := 200;
   Display.Spare3H2 := 0;
   Display.Spare54 := 0;
   Display.Spare55 := 0;
   Display.Spare56 := 0;
   Display.Spare57 := 0;
   Display.Spare58 := 0;
   Display.Overlap2_3 := 100;
   Display.Height3 := -50;
   Display.Landmark3 := TRUE;
   Display.Lifter3 := FALSE;
   Display.SpareBit1H3 := FALSE;
   Display.Airblower3 := TRUE;
   Display.NextStep3 := TRUE;
   Display.PressureP3 := TRUE;
   Display.SpareByte2H3 := 16#00;
   Display.Revolution3 := 2;
   Display.RopeUnit3_1 := 16#01;
   Display.RopeUnit3_2 := 16#01;
   Display.FilmForce3 := 30;
   Display.FilmPrestretch3 := 200;
   Display.Spare3H3 := 0;
   Display.Spare59 := 0;
   Display.Spare60 := 0;
   Display.Spare61 := 380;
   Display.Spare62 := 2800;
   Display.Spare63 := 0;
   Display.Overlap3_4 := 100;
   Display.Height4 := 100;
   Display.Landmark4 := FALSE;
   Display.Lifter4 := FALSE;
   Display.SpareBit1H4 := FALSE;
   Display.Airblower4 := TRUE;
   Display.NextStep4 := TRUE;
   Display.PressureP4 := TRUE;
   Display.SpareByte2H4 := 16#00;
   Display.Revolution4 := 3;
   Display.RopeUnit4_1 := 16#02;
   Display.RopeUnit4_2 := 16#02;
   Display.FilmForce4 := 30;
   Display.FilmPrestretch4 := 200;
   Display.Spare3H4 := 0;
   Display.Spare64 := 0;
   Display.Spare65 := 0;
   Display.Spare66 := 0;
   Display.Spare67 := 0;
   Display.Spare68 := 0;
   Display.Overlap4_5 := 0;
   Display.Height5 := 50;
   Display.Landmark5 := FALSE;
   Display.Lifter5 := FALSE;
   Display.SpareBit1H5 := FALSE;
   Display.Airblower5 := TRUE;
   Display.NextStep5 := FALSE;
   Display.PressureP5 := FALSE;
   Display.SpareByte2H5 := 16#00;
   Display.Revolution5 := 1;
   Display.RopeUnit5_1 := 16#01;
   Display.RopeUnit5_2 := 16#01;
   Display.FilmForce5 := 30;
   Display.FilmPrestretch5 := 200;
   Display.Spare3H5 := 0;
   Display.Spare69 := 0;
   Display.Spare70 := 0;
   Display.Spare71 := 0;
   Display.Spare72 := 0;
   Display.Spare73 := 0;
   Display.Overlap5_6 := 100;
   Display.Height6 := 50;
   Display.Landmark6 := FALSE;
   Display.Lifter6 := FALSE;
   Display.SpareBit1H6 := FALSE;
   Display.Airblower6 := TRUE;
   Display.NextStep6 := FALSE;
   Display.PressureP6 := FALSE;
   Display.SpareByte2H6 := 16#00;
   Display.Revolution6 := 2;
   Display.RopeUnit6_1 := 16#02;
   Display.RopeUnit6_2 := 16#01;
   Display.FilmForce6 := 20;
   Display.FilmPrestretch6 := 200;
   Display.Spare3H6 := 0;
   Display.Spare74 := 0;
   Display.Spare75 := 0;
   Display.Spare76 := 0;
   Display.Spare77 := 0;
   Display.Spare78 := 0;
   Display.Overlap6_7 := 0;
   Display.Height7 := 0;
   Display.Landmark7 := FALSE;
   Display.Lifter7 := FALSE;
   Display.SpareBit1H7 := FALSE;
   Display.Airblower7 := FALSE;
   Display.NextStep7 := TRUE;
   Display.PressureP7 := FALSE;
   Display.SpareByte2H7 := 16#00;
   Display.Revolution7 := 1;
   Display.RopeUnit7_1 := 16#01;
   Display.RopeUnit7_2 := 16#01;
   Display.FilmForce7 := 0;
   Display.FilmPrestretch7 := 100;
   Display.Spare3H7 := 0;
   Display.Spare79 := 0;
   Display.Spare80 := 0;
   Display.Spare81 := 0;
   Display.Spare82 := 0;
   Display.Spare83 := 0;
   Display.Overlap7_8 := 0;
   Display.Height8 := 0;
   Display.Landmark8 := FALSE;
   Display.Lifter8 := FALSE;
   Display.SpareBit1H8 := FALSE;
   Display.Airblower8 := FALSE;
   Display.NextStep8 := TRUE;
   Display.PressureP8 := FALSE;
   Display.SpareByte2H8 := 16#00;
   Display.Revolution8 := 1;
   Display.RopeUnit8_1 := 16#01;
   Display.RopeUnit8_2 := 16#01;
   Display.FilmForce8 := 0;
   Display.FilmPrestretch8 := 100;
   Display.Spare3H8 := 0;
   Display.Spare84 := 0;
   Display.Spare85 := 0;
   Display.Spare86 := 0;
   Display.Spare87 := 0;
   Display.Spare88 := 0;
   Display.Overlap8_9 := 0;
   Display.Height9 := 0;
   Display.Landmark9 := FALSE;
   Display.Lifter9 := FALSE;
   Display.SpareBit1H9 := FALSE;
   Display.Airblower9 := FALSE;
   Display.NextStep9 := TRUE;
   Display.PressureP9 := FALSE;
   Display.SpareByte2H9 := 16#00;
   Display.Revolution9 := 1;
   Display.RopeUnit9_1 := 16#01;
   Display.RopeUnit9_2 := 16#01;
   Display.FilmForce9 := 0;
   Display.FilmPrestretch9 := 100;
   Display.Spare3H9 := 0;
   Display.Spare89 := 0;
   Display.Spare90 := 0;
   Display.Spare91 := 0;
   Display.Spare92 := 0;
   Display.Spare93 := 0;
   Display.Overlap9_10 := 0;
   Display.Height10 := 0;
   Display.Landmark10 := FALSE;
   Display.Lifter10 := FALSE;
   Display.SpareBit1H10 := FALSE;
   Display.Airblower10 := FALSE;
   Display.NextStep10 := FALSE;
   Display.PressureP10 := FALSE;
   Display.SpareByte2H10 := 16#00;
   Display.Revolution10 := 1;
   Display.RopeUnit10_1 := 16#01;
   Display.RopeUnit10_2 := 16#01;
   Display.FilmForce10 := 0;
   Display.FilmPrestretch10 := 100;
   Display.Spare3H10 := 0;
   Display.Spare94 := 0;
   Display.Spare95 := 0;
   Display.Spare96 := 0;
   Display.Spare97 := 0;
   Display.Spare98 := 0;
   Display.Overlap10_11 := 0;
   Display.Height11 := 0;
   Display.Landmark11 := FALSE;
   Display.Lifter11 := FALSE;
   Display.SpareBit1H11 := FALSE;
   Display.Airblower11 := FALSE;
   Display.NextStep11 := TRUE;
   Display.PressureP11 := FALSE;
   Display.SpareByte2H11 := 16#00;
   Display.Revolution11 := 1;
   Display.RopeUnit11_1 := 16#01;
   Display.RopeUnit11_2 := 16#01;
   Display.FilmForce11 := 0;
   Display.FilmPrestretch11 := 100;
   Display.Spare3H11 := 0;
   Display.Spare99 := 0;
   Display.Spare100 := 0;
   Display.Spare101 := 0;
   Display.Spare102 := 0;
   Display.Spare103 := 0;
   Display.Overlap11_12 := 0;
   Display.Height12 := 0;
   Display.Landmark12 := FALSE;
   Display.Lifter12 := FALSE;
   Display.SpareBit1H12 := FALSE;
   Display.Airblower12 := FALSE;
   Display.NextStep12 := FALSE;
   Display.PressureP12 := FALSE;
   Display.SpareByte2H12 := 16#00;
   Display.Revolution12 := 1;
   Display.RopeUnit12_1 := 16#01;
   Display.RopeUnit12_2 := 16#01;
   Display.FilmForce12 := 0;
   Display.FilmPrestretch12 := 100;
   Display.Spare3H12 := 0;
   Display.Spare104 := 0;
   Display.Spare105 := 0;
   Display.Spare106 := 0;
   Display.Spare107 := 0;
   Display.Spare108 := 0;
END_DATA_BLOCK

DATA_BLOCK "DB320_PID"   // DB320
TITLE = PID
{ S7_Optimized_Access := 'FALSE' }
VERSION : 0.1
// stored: AutoNumber false, IsOnlyStoredInLoadMemory false, IsWriteProtectedInAS false
   VAR RETAIN
      PID { S7_SetPoint := 'True'} : "PID";
   END_VAR
BEGIN
   PID.proporzionale := 0;
   PID.integrativo := 0;
   PID.segnale := 0;
   PID.maxSegnale := 1000;
   PID.minSegnale := 0;
   PID.setPointShow := 265;
   PID.tiro := 0;
   PID.vParP := 70;
   PID.vParI := 70;
   PID.svuota := TRUE;
   PID.attiva := TRUE;
   PID.setTiro := FALSE;
   PID."timer" := T#0MS;
END_DATA_BLOCK

DATA_BLOCK "DB322_APP"   // DB322
TITLE = PID
{ S7_Optimized_Access := 'FALSE' }
VERSION : 0.1
// stored: AutoNumber false, IsOnlyStoredInLoadMemory false, IsWriteProtectedInAS false
   VAR RETAIN
      IN0 : Int := 0;
      IN1 : Int := 0;
      IN2 : Int := 0;
      IN3 : Int := 0;
      IN4 : Int := 0;
      IN5 : Int := 0;
      IN6 : Int := 0;
      IN7 : Int := 0;
      IN8 : Int := 0;
      IN9 : Int := 0;
      IN10 : DInt := 224;
      IN11 : DInt := 240;
      IN12 : DInt := 0;   // TIRO EQUIVALENTE SU CELLA (kg)
      APP { S7_SetPoint := 'True'} : "APP";
   END_VAR
BEGIN
   APP.PID_ComponenteProporzionale := 0;
   APP.PID_ComponenteIntegrale := 0;
   APP.PID_ComponenteDerivativa := 0;
   APP.Tiro := 0;
   APP.Tiro1 := 0;
   APP.Tiro2 := 0;
   APP.TiroPrecedente := 0;
   APP.TiroAppoggio := 0;
   APP.ErroreAttuale := 0;
   APP.ErrorePrecedente := 0;
   APP.PID_Kp := 70;
   APP.PID_Ki := 60;
   APP.PID_Kd := 0;
   APP.SetpointTiro := 56;
   APP.SetpointTiroRampa := 750;
   APP.TransitorioInizialeFase1 := 0;
   APP.TransitorioFase3 := 1;
   APP.TransitorioFase4 := 1;
   APP.VelocitaRotazione := 5;
   APP.VelocitaRotazioneFase2 := 100;
   APP.VelocitaRotazioneAppoggio1 := 100;
   APP.VelocitaRotazioneAppoggio2 := 100;
   APP.Fase1OneShoot := 0;
   APP.Fase2OneShoot := 0;
   APP.Fase3OneShoot := 0;
   APP.Fase4OneShoot := 0;
   APP.ArrestoRepentinoOneShoot := 0;
   APP.TiroFase1 := 0;
   APP.TempIntero := 90;
   APP.Fase := 0;
   APP.BallerinoPrecedente[0..2] := 56;
   APP.LimiteComponenteIntegrale := 20000;
   APP.TiroRichiesto := 10;
   APP.TimerArrestoRepentino := 2;
   APP.TiroMinimoArrestoRepentino := 10;
   APP.VariazioneTiro := 0;
   APP.TimerFase2 := 0;
   APP.TempoRotturaFilm := 166;
   APP.TimerFase4 := 0;
   APP.TiroMinimoFase4 := 6;
   APP.PID_Uscita := 0;
   APP.PrestiroRichiesto := 300;
   APP.PrestiroAppoggio := 0.5;
END_DATA_BLOCK

DATA_BLOCK "DB50_Config"   // DB50
{ S7_Optimized_Access := 'FALSE' }
VERSION : 0.1
// stored: AutoNumber false, IsOnlyStoredInLoadMemory false, IsWriteProtectedInAS false
   VAR RETAIN
      Sel1_Clamp : Int := 3;
      Sel2_BarrierIn : Int := 2;
      Sel3_Pressure : Int := 1;
      Sel4_Doors : Int := 0;
      Sel5_Carriage : Int := 1;
      Sel6_Selfcenter : Int := 2;
      Sel7_Top : Int := 1;
      Sel8_Rope : Int := 3;
      Sel9_BarrierOut : Int := 2;
      Sel10_Conv : Int := 16;
      Sel_Door : Bool := TRUE;
      Sel_EsaurFilm : Bool := FALSE;
      Sel_spare_bool_1 : Bool := FALSE;
      Sel_spare_bool_2 : Bool := FALSE;
      Sel_spare_bool_3 : Bool := FALSE;
      Sel_spare_bool_4 : Bool := FALSE;
      Sel_spare_bool_5 : Bool := FALSE;
      Sel_spare10 : Byte := 16#00;
      Sel_spare11 : Int := 0;
      Sel_spare12 : Int := 0;
      Sel_spare13 : Int := 0;
      Sel_spare14 : Int := 0;
      Sel_spare15 : Int := 0;
      Sel_spare16 : Int := 0;
      Sel_spare17 : Int := 0;
      Sel_spare18 : Int := 0;
      Sel_spare19 : Int := 0;
      Sel_spare20 : Int := 0;
      Sel_spare21 : Int := 0;
      Sel_spare22 : Int := 0;
      Sel_spare23 : Int := 0;
      Sel_spare24 : Int := 0;
      TimerPageFw : Bool := FALSE;
      TimerPageBkw : Bool := FALSE;
   END_VAR
BEGIN
END_DATA_BLOCK

DATA_BLOCK "DB80_Label"   // DB80
{ S7_Optimized_Access := 'FALSE' }
VERSION : 0.1
// stored: AutoNumber false, IsOnlyStoredInLoadMemory false, IsWriteProtectedInAS false
   VAR RETAIN
      Step0 : Bool := FALSE;   // Table rotation to first label position
      Step1 : Bool := FALSE;   // First label apply
      Step2 : Bool := FALSE;   // Table rotation to second label position
      Step3 : Bool := FALSE;   // Second label apply
      Step4 : Bool := FALSE;   // Table rotation to third label position
      Step5 : Bool := FALSE;   // Third label apply
      Step6 : Bool := FALSE;   // Table rotation to fourth label position
      Step7 : Bool := FALSE;   // Fourt label apply
      Step8 : Bool := FALSE;   // Table rotation to end cycle position
      spare_Step9 : Bool := FALSE;
      spare_Step10 : Bool := FALSE;
      spare_Step11 : Bool := FALSE;
      spare_Step12 : Bool := FALSE;
      spare_Step13 : Bool := FALSE;
      spare_Step14 : Bool := FALSE;
      spare_Step15 : Bool := FALSE;
      Phase1_On : Bool := TRUE;
      Phase2_On : Bool := FALSE;
      Phase3_On : Bool := TRUE;
      Phase4_On : Bool := FALSE;
      Enable : Bool := TRUE;
      rotation : Bool := FALSE;   // Table rotation for label command
      label_ok1 : Bool := FALSE;   // Label cycle ended
      S1 : Bool := FALSE;   // Label request signal
      spare_signal2 : Bool := FALSE;
      spare_signal3 : Bool := FALSE;
      spare_signal4 : Bool := FALSE;
      spare_signal5 : Bool := FALSE;
      spare_signal6 : Bool := FALSE;
      spare_signal7 : Bool := FALSE;
      spare_signal8 : Bool := FALSE;
      E1 : Bool := TRUE;   // Label arm in home position for pallet transit
      E2 : Bool := FALSE;   // Label applied signal
      E3 : Bool := FALSE;   // Label fault signal
      spare_input4 : Bool := FALSE;
      spare_input5 : Bool := FALSE;
      spare_input6 : Bool := FALSE;
      spare_input7 : Bool := FALSE;
      spare_input8 : Bool := FALSE;
      spare_byte5 : Byte := 16#00;
      Phase1 : Int := 900;
      Phase2 : Int := 1800;
      Phase3 : Int := 2700;
      Phase4 : Int := 3600;
      NextPhase : Int := 2700;
   END_VAR
BEGIN
END_DATA_BLOCK

DATA_BLOCK "DB88_Top"   // DB88
{ S7_Optimized_Access := 'FALSE' }
AUTHOR : Robopac
VERSION : 0.0
// stored: AutoNumber false, IsOnlyStoredInLoadMemory false, IsWriteProtectedInAS false
   VAR RETAIN
      VW800 : Int := 0;
      VW802 : Int := 0;
      V804_0 : Bool := FALSE;   // Top carriage in cut position
      V804_1 : Bool := FALSE;   // Top carriage in forward position
      V804_2 : Bool := FALSE;
      V804_3 : Bool := FALSE;   // Memory to stop top carriage forward in manual mode
      V804_4 : Bool := FALSE;   // Memory for top cut done
      V804_5 : Bool := FALSE;
      V804_6 : Bool := FALSE;
      V804_7 : Bool := FALSE;
      VB805 : Byte := 16#00;
      VW806 : Int := 0;   // Top positioning counter
   END_VAR
BEGIN
END_DATA_BLOCK

DATA_BLOCK "DeviceStates"   // DB12
{ S7_Optimized_Access := 'FALSE' }
VERSION : 0.1
// stored: AutoNumber true, IsOnlyStoredInLoadMemory false, IsWriteProtectedInAS false
   VAR
      LADDR : HW_IOSYSTEM := 16#010F;
      MODE : UInt := 4;
      returnValue : Int := 0;
      STATE : Array[0..1023] of Bool;
   END_VAR
BEGIN
   STATE[0..3] := TRUE;
   STATE[4..1023] := FALSE;
END_DATA_BLOCK

DATA_BLOCK "Inverter_Data"   // DB210
{ S7_Optimized_Access := 'FALSE' }
VERSION : 0.1
// stored: AutoNumber false, IsOnlyStoredInLoadMemory false, IsWriteProtectedInAS false
   VAR
      U201 { S7_SetPoint := 'True'} : "InverterData";
      U221 { S7_SetPoint := 'True'} : "InverterData";
      U241 { S7_SetPoint := 'True'} : "InverterData";
      U261 { S7_SetPoint := 'True'} : "InverterData";
      U321 { S7_SetPoint := 'True'} : "InverterData";
   END_VAR
BEGIN
   U201.control_word := 16#047A;
   U201.setpoint := 0.0;
   U201.ref_quantity.speed_p2000 := 3000.0;
   U201.ref_quantity.current_p2002 := 5.0;
   U201.ref_quantity.torque_p2003 := 7.61;
   U201.status_word := 16#EB40;
   U201.actual_speed := 0.0;
   U201.actual_current := 0.0;
   U201.actual_torque := 0.0;
   U201.actual_alarm := 16#0000;
   U201.actual_fault := 16#0000;
   U201.RETVAL_RD := 16#0000;
   U201.RETVAL_WR := 16#0000;
   U221.control_word := 16#047E;
   U221.setpoint := 0.0;
   U221.ref_quantity.speed_p2000 := 3000.0;
   U221.ref_quantity.current_p2002 := 1.86;
   U221.ref_quantity.torque_p2003 := 3.59;
   U221.status_word := 16#EB31;
   U221.actual_speed := 0.0;
   U221.actual_current := 0.001702881;
   U221.actual_torque := 0.0;
   U221.actual_alarm := 16#0000;
   U221.actual_fault := 16#0000;
   U221.RETVAL_RD := 16#0000;
   U221.RETVAL_WR := 16#0000;
   U241.control_word := 16#047E;
   U241.setpoint := 0.0;
   U241.ref_quantity.speed_p2000 := 3000.0;
   U241.ref_quantity.current_p2002 := 1.86;
   U241.ref_quantity.torque_p2003 := 3.59;
   U241.status_word := 16#EB31;
   U241.actual_speed := 0.0;
   U241.actual_current := 0.002043457;
   U241.actual_torque := 0.0;
   U241.actual_alarm := 16#0000;
   U241.actual_fault := 16#0000;
   U241.RETVAL_RD := 16#0000;
   U241.RETVAL_WR := 16#0000;
   U261.control_word := 16#047E;
   U261.setpoint := 0.0;
   U261.ref_quantity.speed_p2000 := 3000.0;
   U261.ref_quantity.current_p2002 := 1.86;
   U261.ref_quantity.torque_p2003 := 3.59;
   U261.status_word := 16#EB31;
   U261.actual_speed := 0.0;
   U261.actual_current := 0.0;
   U261.actual_torque := 0.0;
   U261.actual_alarm := 16#0000;
   U261.actual_fault := 16#0000;
   U261.RETVAL_RD := 16#0000;
   U261.RETVAL_WR := 16#0000;
   U321.control_word := 16#047E;
   U321.setpoint := 0.0;
   U321.ref_quantity.speed_p2000 := 3000.0;
   U321.ref_quantity.current_p2002 := 6.9;
   U321.ref_quantity.torque_p2003 := 29.5;
   U321.status_word := 16#EB31;
   U321.actual_speed := 0.0;
   U321.actual_current := 0.0;
   U321.actual_torque := 0.0;
   U321.actual_alarm := 16#0000;
   U321.actual_fault := 16#0000;
   U321.RETVAL_RD := 16#0000;
   U321.RETVAL_WR := 16#0000;
END_DATA_BLOCK

